LIN {X 0,Y 301.747,Z 438.159,A -85,B 0,C 180,E1 -16541.674,E2 -16541.674} C_VEL
LIN {X 0,Y 303.087,Z 433.963,A -85,B 0,C 180,E1 -16543.844,E2 -16543.844} C_VEL
LIN {X 0,Y 304.497,Z 429.034,A -85,B 0,C 180,E1 -16545.781,E2 -16545.781} C_VEL
LIN {X 0,Y 306.519,Z 421.411,A -85,B 0,C 180,E1 -16548.091,E2 -16548.091} C_VEL
LIN {X 0,Y 308.265,Z 414.22,A -85,B 0,C 180,E1 -16549.823,E2 -16549.823} C_VEL
LIN {X 0,Y 310.172,Z 405.497,A -85,B 0,C 180,E1 -16551.531,E2 -16551.531} C_VEL
LIN {X 0,Y 312.108,Z 395.019,A -85,B 0,C 180,E1 -16553.171,E2 -16553.171} C_VEL
LIN {X 0,Y 312.343,Z 393.686,A -85,B 0,C 180,E1 -16553.358,E2 -16553.358} C_VEL
LIN {X 0,Y 310.159,Z 384.516,A -85,B 0,C 180,E1 -16554.99,E2 -16554.99} C_VEL
LIN {X 0,Y 307.115,Z 376.232,A -85,B 0,C 180,E1 -16556.443,E2 -16556.443} C_VEL
LIN {X 0,Y 305.388,Z 373.91,A -85,B 0,C 180,E1 -16556.951,E2 -16556.951} C_VEL
LIN {X 0,Y 301.445,Z 371.285,A -85,B 0,C 180,E1 -16557.846,E2 -16557.846} C_VEL
LIN {X 0,Y 297.397,Z 368.735,A -85,B 0,C 180,E1 -16558.76,E2 -16558.76} C_VEL
LIN {X 0,Y 295.474,Z 366.51,A -85,B 0,C 180,E1 -16559.287,E2 -16559.287} C_VEL
LIN {X 0,Y 292.034,Z 359.85,A -85,B 0,C 180,E1 -16560.517,E2 -16560.517} C_VEL
LIN {X 0,Y 291.896,Z 359.149,A -85,B 0,C 180,E1 -16560.949,E2 -16560.949} C_VEL
LIN {X 0,Y 291.539,Z 359.172,A -85,B 0,C 180,E1 -16564.147,E2 -16564.147} C_VEL
LIN {X 0,Y 291.714,Z 359.147,A -85,B 0,C 180,E1 -16566.919,E2 -16566.919} C_VEL
LIN {X 0,Y 291.561,Z 359.165,A -85,B 0,C 180,E1 -16569.714,E2 -16569.714} C_VEL
LIN {X 0,Y 291.508,Z 359.173,A -85,B 0,C 180,E1 -16573.951,E2 -16573.951} C_VEL
LIN {X 0,Y 291.426,Z 359.18,A -85,B 0,C 180,E1 -16576.822,E2 -16576.822} C_VEL
LIN {X 0,Y 291.418,Z 359.182,A -85,B 0,C 180,E1 -16579.861,E2 -16579.861} C_VEL
LIN {X 0,Y 291.376,Z 359.185,A -85,B 0,C 180,E1 -16584.208,E2 -16584.208} C_VEL
LIN {X 0,Y 291.413,Z 359.184,A -85,B 0,C 180,E1 -16587.273,E2 -16587.273} C_VEL
LIN {X 0,Y 291.329,Z 359.196,A -85,B 0,C 180,E1 -16590.438,E2 -16590.438} C_VEL
LIN {X 0,Y 291.381,Z 359.44,A -85,B 0,C 180,E1 -16593.337,E2 -16593.337} C_VEL
LIN {X 0,Y 292.227,Z 363.097,A -85,B 0,C 180,E1 -16596.959,E2 -16596.959} C_VEL
LIN {X 0,Y 293.339,Z 368.291,A -85,B 0,C 180,E1 -16601.213,E2 -16601.213} C_VEL
LIN {X 0,Y 294.41,Z 373.527,A -85,B 0,C 180,E1 -16604.848,E2 -16604.848} C_VEL
LIN {X 0,Y 295.479,Z 379.098,A -85,B 0,C 180,E1 -16608.244,E2 -16608.244} C_VEL
LIN {X 0,Y 296.242,Z 383.983,A -85,B 0,C 180,E1 -16610.941,E2 -16610.941} C_VEL
LIN {X 0,Y 296.147,Z 385.908,A -85,B 0,C 180,E1 -16611.902,E2 -16611.902} C_VEL
LIN {X 0,Y 294.347,Z 394.571,A -85,B 0,C 180,E1 -16615.869,E2 -16615.869} C_VEL
LIN {X 0,Y 292.656,Z 405.269,A -85,B 0,C 180,E1 -16620.509,E2 -16620.509} C_VEL
LIN {X 0,Y 292.601,Z 406.741,A -85,B 0,C 180,E1 -16620.947,E2 -16620.947} C_VEL
LIN {X 0,Y 296.051,Z 421.846,A -85,B 0,C 180,E1 -16622.426,E2 -16622.426} C_VEL
LIN {X 0,Y 298.005,Z 434.056,A -85,B 0,C 180,E1 -16623.66,E2 -16623.66} C_VEL
LIN {X 0,Y 298.946,Z 446.03,A -85,B 0,C 180,E1 -16624.966,E2 -16624.966} C_VEL
LIN {X 0,Y 298.863,Z 458.909,A -85,B 0,C 180,E1 -16626.508,E2 -16626.508} C_VEL
LIN {X 0,Y 297.735,Z 470.963,A -85,B 0,C 180,E1 -16628.175,E2 -16628.175} C_VEL
LIN {X 0,Y 296.455,Z 481.364,A -85,B 0,C 180,E1 -16629.895,E2 -16629.895} C_VEL
LIN {X 0,Y 294.247,Z 491.64,A -85,B 0,C 180,E1 -16631.911,E2 -16631.911} C_VEL
LIN {X 0,Y 292.426,Z 500.348,A -85,B 0,C 180,E1 -16634.016,E2 -16634.016} C_VEL
LIN {X 0,Y 291.545,Z 506.044,A -85,B 0,C 180,E1 -16635.695,E2 -16635.695} C_VEL
LIN {X 0,Y 290.556,Z 512.87,A -85,B 0,C 180,E1 -16638.136,E2 -16638.136} C_VEL
LIN {X 0,Y 290.137,Z 517.474,A -85,B 0,C 180,E1 -16640.238,E2 -16640.238} C_VEL
LIN {X 0,Y 290.167,Z 521.068,A -85,B 0,C 180,E1 -16642.345,E2 -16642.345} C_VEL
LIN {X 0,Y 290.425,Z 523.677,A -85,B 0,C 180,E1 -16644.445,E2 -16644.445} C_VEL
LIN {X 0,Y 290.726,Z 524.917,A -85,B 0,C 180,E1 -16645.841,E2 -16645.841} C_VEL
LIN {X 0,Y 291.329,Z 526.05,A -85,B 0,C 180,E1 -16648.618,E2 -16648.618} C_VEL
LIN {X 0,Y 291.637,Z 525.995,A -85,B 0,C 180,E1 -16650,E2 -16650} C_VEL
LIN {X 0,Y 291.369,Z 525.423,A -85,B 0,C 180,E1 -16651.382,E2 -16651.382} C_VEL
LIN {X 0,Y 291.047,Z 524.355,A -85,B 0,C 180,E1 -16652.768,E2 -16652.768} C_VEL
LIN {X 0,Y 290.904,Z 522.87,A -85,B 0,C 180,E1 -16654.156,E2 -16654.156} C_VEL
LIN {X 0,Y 290.642,Z 519.728,A -85,B 0,C 180,E1 -16656.247,E2 -16656.247} C_VEL
LIN {X 0,Y 290.456,Z 515.429,A -85,B 0,C 180,E1 -16658.347,E2 -16658.347} C_VEL
LIN {X 0,Y 290.489,Z 509.882,A -85,B 0,C 180,E1 -16660.454,E2 -16660.454} C_VEL
LIN {X 0,Y 290.897,Z 502.911,A -85,B 0,C 180,E1 -16662.558,E2 -16662.558} C_VEL
LIN {X 0,Y 291.721,Z 494.208,A -85,B 0,C 180,E1 -16664.652,E2 -16664.652} C_VEL
LIN {X 0,Y 292.782,Z 485.266,A -85,B 0,C 180,E1 -16666.399,E2 -16666.399} C_VEL
LIN {X 0,Y 293.913,Z 475.665,A -85,B 0,C 180,E1 -16667.93,E2 -16667.93} C_VEL
LIN {X 0,Y 293.764,Z 463.078,A -85,B 0,C 180,E1 -16669.568,E2 -16669.568} C_VEL
LIN {X 0,Y 293.258,Z 451.021,A -85,B 0,C 180,E1 -16670.828,E2 -16670.828} C_VEL
LIN {X 0,Y 292.555,Z 438.329,A -85,B 0,C 180,E1 -16671.86,E2 -16671.86} C_VEL
LIN {X 0,Y 291.466,Z 424.734,A -85,B 0,C 180,E1 -16672.693,E2 -16672.693} C_VEL
LIN {X 0,Y 290.934,Z 418.518,A -85,B 0,C 180,E1 -16673.031,E2 -16673.031} C_VEL
LIN {X 0,Y 291.153,Z 415.339,A -85,B 0,C 180,E1 -16674.226,E2 -16674.226} C_VEL
LIN {X 0,Y 292.285,Z 404.281,A -85,B 0,C 180,E1 -16678.743,E2 -16678.743} C_VEL
LIN {X 0,Y 293.696,Z 393.683,A -85,B 0,C 180,E1 -16683.119,E2 -16683.119} C_VEL
LIN {X 0,Y 295.372,Z 383.621,A -85,B 0,C 180,E1 -16687.353,E2 -16687.353} C_VEL
LIN {X 0,Y 295.557,Z 381.391,A -85,B 0,C 180,E1 -16688.307,E2 -16688.307} C_VEL
LIN {X 0,Y 294.425,Z 374.995,A -85,B 0,C 180,E1 -16691.223,E2 -16691.223} C_VEL
LIN {X 0,Y 292.932,Z 367.204,A -85,B 0,C 180,E1 -16694.947,E2 -16694.947} C_VEL
LIN {X 0,Y 291.334,Z 359.27,A -85,B 0,C 180,E1 -16698.995,E2 -16698.995} C_VEL
LIN {X 0,Y 291.396,Z 359.188,A -85,B 0,C 180,E1 -16702.918,E2 -16702.918} C_VEL
LIN {X 0,Y 291.34,Z 359.192,A -85,B 0,C 180,E1 -16706.301,E2 -16706.301} C_VEL
LIN {X 0,Y 291.382,Z 359.186,A -85,B 0,C 180,E1 -16710.26,E2 -16710.26} C_VEL
LIN {X 0,Y 291.405,Z 359.184,A -85,B 0,C 180,E1 -16714.271,E2 -16714.271} C_VEL
LIN {X 0,Y 291.366,Z 359.191,A -85,B 0,C 180,E1 -16717.298,E2 -16717.298} C_VEL
LIN {X 0,Y 291.433,Z 359.18,A -85,B 0,C 180,E1 -16720.268,E2 -16720.268} C_VEL
LIN {X 0,Y 291.491,Z 359.175,A -85,B 0,C 180,E1 -16724.665,E2 -16724.665} C_VEL
LIN {X 0,Y 291.521,Z 359.172,A -85,B 0,C 180,E1 -16728.88,E2 -16728.88} C_VEL
LIN {X 0,Y 291.659,Z 359.152,A -85,B 0,C 180,E1 -16731.687,E2 -16731.687} C_VEL
LIN {X 0,Y 291.61,Z 359.16,A -85,B 0,C 180,E1 -16734.468,E2 -16734.468} C_VEL
LIN {X 0,Y 291.881,Z 359.127,A -85,B 0,C 180,E1 -16738.62,E2 -16738.62} C_VEL
LIN {X 0,Y 291.881,Z 359.125,A -85,B 0,C 180,E1 -16741.38,E2 -16741.38} C_VEL
LIN {X 0,Y 291.734,Z 359.146,A -85,B 0,C 180,E1 -16746.918,E2 -16746.918} C_VEL
LIN {X 0,Y 291.622,Z 359.156,A -85,B 0,C 180,E1 -16749.712,E2 -16749.712} C_VEL
LIN {X 0,Y 291.515,Z 359.169,A -85,B 0,C 180,E1 -16753.951,E2 -16753.951} C_VEL
LIN {X 0,Y 291.48,Z 359.177,A -85,B 0,C 180,E1 -16756.818,E2 -16756.818} C_VEL
LIN {X 0,Y 291.445,Z 359.179,A -85,B 0,C 180,E1 -16759.875,E2 -16759.875} C_VEL
LIN {X 0,Y 291.394,Z 359.187,A -85,B 0,C 180,E1 -16764.206,E2 -16764.206} C_VEL
LIN {X 0,Y 291.417,Z 359.182,A -85,B 0,C 180,E1 -16767.272,E2 -16767.272} C_VEL
LIN {X 0,Y 291.332,Z 359.197,A -85,B 0,C 180,E1 -16770.437,E2 -16770.437} C_VEL
LIN {X 0,Y 291.34,Z 359.192,A -85,B 0,C 180,E1 -16773.699,E2 -16773.699} C_VEL
LIN {X 0,Y 291.393,Z 359.184,A -85,B 0,C 180,E1 -16777.26,E2 -16777.26} C_VEL
LIN {X 0,Y 291.372,Z 359.19,A -85,B 0,C 180,E1 -16780.636,E2 -16780.636} C_VEL
LIN {X 0,Y 291.297,Z 359.2,A -85,B 0,C 180,E1 -16784.401,E2 -16784.401} C_VEL
LIN {X 0,Y 291.324,Z 359.196,A -85,B 0,C 180,E1 -16788.405,E2 -16788.405} C_VEL
LIN {X 0,Y 291.362,Z 359.189,A -85,B 0,C 180,E1 -16791.161,E2 -16791.161} C_VEL
LIN {X 0,Y 291.361,Z 359.189,A -85,B 0,C 180,E1 -16794.627,E2 -16794.627} C_VEL
LIN {X 0,Y 291.375,Z 359.192,A -85,B 0,C 180,E1 -16797.952,E2 -16797.952} C_VEL
LIN {X 0,Y 291.387,Z 359.186,A -85,B 0,C 180,E1 -16801.16,E2 -16801.16} C_VEL
LIN {X 0,Y 291.418,Z 359.184,A -85,B 0,C 180,E1 -16804.273,E2 -16804.273} C_VEL
LIN {X 0,Y 291.382,Z 359.187,A -85,B 0,C 180,E1 -16807.3,E2 -16807.3} C_VEL
LIN {X 0,Y 291.459,Z 359.178,A -85,B 0,C 180,E1 -16810.271,E2 -16810.271} C_VEL
LIN {X 0,Y 291.556,Z 359.165,A -85,B 0,C 180,E1 -16814.624,E2 -16814.624} C_VEL
LIN {X 0,Y 291.539,Z 359.166,A -85,B 0,C 180,E1 -16818.881,E2 -16818.881} C_VEL
LIN {X 0,Y 291.712,Z 359.15,A -85,B 0,C 180,E1 -16821.689,E2 -16821.689} C_VEL
LIN {X 0,Y 291.634,Z 359.155,A -85,B 0,C 180,E1 -16824.469,E2 -16824.469} C_VEL
LIN {X 0,Y 291.895,Z 359.122,A -85,B 0,C 180,E1 -16828.62,E2 -16828.62} C_VEL
LIN {X 0,Y 291.892,Z 359.127,A -85,B 0,C 180,E1 -16831.38,E2 -16831.38} C_VEL
LIN {X 0,Y 291.738,Z 359.143,A -85,B 0,C 180,E1 -16836.918,E2 -16836.918} C_VEL
LIN {X 0,Y 291.63,Z 359.158,A -85,B 0,C 180,E1 -16839.712,E2 -16839.712} C_VEL
LIN {X 0,Y 291.524,Z 359.17,A -85,B 0,C 180,E1 -16843.95,E2 -16843.95} C_VEL
LIN {X 0,Y 291.488,Z 359.174,A -85,B 0,C 180,E1 -16846.817,E2 -16846.817} C_VEL
LIN {X 0,Y 291.451,Z 359.179,A -85,B 0,C 180,E1 -16849.874,E2 -16849.874} C_VEL
LIN {X 0,Y 291.399,Z 359.184,A -85,B 0,C 180,E1 -16854.205,E2 -16854.205} C_VEL
LIN {X 0,Y 291.418,Z 359.186,A -85,B 0,C 180,E1 -16857.271,E2 -16857.271} C_VEL
LIN {X 0,Y 291.333,Z 359.193,A -85,B 0,C 180,E1 -16860.436,E2 -16860.436} C_VEL
LIN {X 0,Y 291.343,Z 359.193,A -85,B 0,C 180,E1 -16863.698,E2 -16863.698} C_VEL
LIN {X 0,Y 291.404,Z 359.188,A -85,B 0,C 180,E1 -16867.261,E2 -16867.261} C_VEL
LIN {X 0,Y 291.463,Z 359.34,A -85,B 0,C 180,E1 -16870.445,E2 -16870.445} C_VEL
LIN {X 0,Y 291.684,Z 360.374,A -85,B 0,C 180,E1 -16870.68,E2 -16870.68} C_VEL
LIN {X 0,Y 295.511,Z 373.533,A -85,B 0,C 180,E1 -16872.122,E2 -16872.122} C_VEL
LIN {X 0,Y 297.723,Z 381.938,A -85,B 0,C 180,E1 -16873.2,E2 -16873.2} C_VEL
LIN {X 0,Y 297.506,Z 387.452,A -85,B 0,C 180,E1 -16873.904,E2 -16873.904} C_VEL
LIN {X 0,Y 296.304,Z 399.361,A -85,B 0,C 180,E1 -16875.658,E2 -16875.658} C_VEL
LIN {X 0,Y 295.192,Z 408.983,A -85,B 0,C 180,E1 -16877.423,E2 -16877.423} C_VEL
LIN {X 0,Y 294.133,Z 417.653,A -85,B 0,C 180,E1 -16879.375,E2 -16879.375} C_VEL
LIN {X 0,Y 293.327,Z 425.193,A -85,B 0,C 180,E1 -16881.468,E2 -16881.468} C_VEL
LIN {X 0,Y 292.501,Z 432.164,A -85,B 0,C 180,E1 -16883.937,E2 -16883.937} C_VEL
LIN {X 0,Y 292.005,Z 437.44,A -85,B 0,C 180,E1 -16886.388,E2 -16886.388} C_VEL
LIN {X 0,Y 291.744,Z 441.153,A -85,B 0,C 180,E1 -16888.807,E2 -16888.807} C_VEL
LIN {X 0,Y 291.721,Z 443.554,A -85,B 0,C 180,E1 -16891.195,E2 -16891.195} C_VEL
LIN {X 0,Y 291.842,Z 444.59,A -85,B 0,C 180,E1 -16892.998,E2 -16892.998} C_VEL
LIN {X 0,Y 292.048,Z 444.896,A -85,B 0,C 180,E1 -16894.332,E2 -16894.332} C_VEL
LIN {X 0,Y 292.447,Z 444.8,A -85,B 0,C 180,E1 -16895.949,E2 -16895.949} C_VEL
LIN {X 0,Y 292.9,Z 444.204,A -85,B 0,C 180,E1 -16897.424,E2 -16897.424} C_VEL
LIN {X 0,Y 293.512,Z 443.042,A -85,B 0,C 180,E1 -16899.037,E2 -16899.037} C_VEL
LIN {X 0,Y 294.518,Z 440.572,A -85,B 0,C 180,E1 -16901.207,E2 -16901.207} C_VEL
LIN {X 0,Y 295.861,Z 436.851,A -85,B 0,C 180,E1 -16903.438,E2 -16903.438} C_VEL
LIN {X 0,Y 297.42,Z 431.843,A -85,B 0,C 180,E1 -16905.65,E2 -16905.65} C_VEL
LIN {X 0,Y 299.307,Z 425.489,A -85,B 0,C 180,E1 -16907.8,E2 -16907.8} C_VEL
LIN {X 0,Y 301.082,Z 418.897,A -85,B 0,C 180,E1 -16909.58,E2 -16909.58} C_VEL
LIN {X 0,Y 303.008,Z 410.961,A -85,B 0,C 180,E1 -16911.329,E2 -16911.329} C_VEL
LIN {X 0,Y 305.084,Z 401.311,A -85,B 0,C 180,E1 -16913.036,E2 -16913.036} C_VEL
LIN {X 0,Y 305.93,Z 396.746,A -85,B 0,C 180,E1 -16913.736,E2 -16913.736} C_VEL
LIN {X 0,Y 305.723,Z 393.97,A -85,B 0,C 180,E1 -16914.234,E2 -16914.234} C_VEL
LIN {X 0,Y 303.779,Z 386.226,A -85,B 0,C 180,E1 -16915.688,E2 -16915.688} C_VEL
LIN {X 0,Y 300.007,Z 376.53,A -85,B 0,C 180,E1 -16917.499,E2 -16917.499} C_VEL
LIN {X 0,Y 295.799,Z 367.062,A -85,B 0,C 180,E1 -16919.181,E2 -16919.181} C_VEL
LIN {X 0,Y 295.474,Z 366.51,A -85,B 0,C 180,E1 -16919.287,E2 -16919.287} C_VEL
LIN {X 0,Y 293.577,Z 364.13,A -85,B 0,C 180,E1 -16919.839,E2 -16919.839} C_VEL
LIN {X 0,Y 289.506,Z 361.509,A -85,B 0,C 180,E1 -16920.824,E2 -16920.824} C_VEL
LIN {X 0,Y 286.336,Z 360.394,A -85,B 0,C 180,E1 -16921.682,E2 -16921.682} C_VEL
LIN {X 0,Y 284.881,Z 360.039,A -85,B 0,C 180,E1 -16922.422,E2 -16922.422} C_VEL
LIN {X 0,Y 284.743,Z 360.017,A -85,B 0,C 180,E1 -16922.687,E2 -16922.687} C_VEL
LIN {X 0,Y 284.665,Z 360.026,A -85,B 0,C 180,E1 -16927.091,E2 -16927.091} C_VEL
LIN {X 0,Y 284.507,Z 360.044,A -85,B 0,C 180,E1 -16929.958,E2 -16929.958} C_VEL
LIN {X 0,Y 284.456,Z 360.053,A -85,B 0,C 180,E1 -16934.304,E2 -16934.304} C_VEL
LIN {X 0,Y 284.356,Z 360.062,A -85,B 0,C 180,E1 -16938.742,E2 -16938.742} C_VEL
LIN {X 0,Y 284.309,Z 360.068,A -85,B 0,C 180,E1 -16941.765,E2 -16941.765} C_VEL
LIN {X 0,Y 284.33,Z 360.068,A -85,B 0,C 180,E1 -16944.847,E2 -16944.847} C_VEL
LIN {X 0,Y 284.322,Z 360.068,A -85,B 0,C 180,E1 -16948.012,E2 -16948.012} C_VEL
LIN {X 0,Y 284.322,Z 360.288,A -85,B 0,C 180,E1 -16951.683,E2 -16951.683} C_VEL
LIN {X 0,Y 285.149,Z 363.846,A -85,B 0,C 180,E1 -16955.578,E2 -16955.578} C_VEL
LIN {X 0,Y 286.14,Z 368.455,A -85,B 0,C 180,E1 -16959.687,E2 -16959.687} C_VEL
LIN {X 0,Y 287.406,Z 374.342,A -85,B 0,C 180,E1 -16964.057,E2 -16964.057} C_VEL
LIN {X 0,Y 288.542,Z 380.473,A -85,B 0,C 180,E1 -16967.962,E2 -16967.962} C_VEL
LIN {X 0,Y 289.336,Z 385.842,A -85,B 0,C 180,E1 -16971.013,E2 -16971.013} C_VEL
LIN {X 0,Y 288.834,Z 388.945,A -85,B 0,C 180,E1 -16972.534,E2 -16972.534} C_VEL
LIN {X 0,Y 286.927,Z 398.192,A -85,B 0,C 180,E1 -16976.845,E2 -16976.845} C_VEL
LIN {X 0,Y 285.916,Z 404.822,A -85,B 0,C 180,E1 -16979.691,E2 -16979.691} C_VEL
LIN {X 0,Y 286.502,Z 408.028,A -85,B 0,C 180,E1 -16980.074,E2 -16980.074} C_VEL
LIN {X 0,Y 289.27,Z 418.993,A -85,B 0,C 180,E1 -16981.228,E2 -16981.228} C_VEL
LIN {X 0,Y 291.495,Z 433.005,A -85,B 0,C 180,E1 -16982.737,E2 -16982.737} C_VEL
LIN {X 0,Y 292.615,Z 446.26,A -85,B 0,C 180,E1 -16984.261,E2 -16984.261} C_VEL
LIN {X 0,Y 292.378,Z 458.983,A -85,B 0,C 180,E1 -16985.882,E2 -16985.882} C_VEL
LIN {X 0,Y 291.136,Z 471.212,A -85,B 0,C 180,E1 -16987.654,E2 -16987.654} C_VEL
LIN {X 0,Y 289.735,Z 481.334,A -85,B 0,C 180,E1 -16989.408,E2 -16989.408} C_VEL
LIN {X 0,Y 287.824,Z 489.848,A -85,B 0,C 180,E1 -16991.124,E2 -16991.124} C_VEL
LIN {X 0,Y 285.862,Z 498.805,A -85,B 0,C 180,E1 -16993.328,E2 -16993.328} C_VEL
LIN {X 0,Y 284.389,Z 506.549,A -85,B 0,C 180,E1 -16995.693,E2 -16995.693} C_VEL
LIN {X 0,Y 283.539,Z 512.172,A -85,B 0,C 180,E1 -16997.838,E2 -16997.838} C_VEL
LIN {X 0,Y 283.086,Z 516.691,A -85,B 0,C 180,E1 -16999.992,E2 -16999.992} C_VEL
LIN {X 0,Y 283.185,Z 521.141,A -85,B 0,C 180,E1 -17002.872,E2 -17002.872} C_VEL
LIN {X 0,Y 283.336,Z 522.751,A -85,B 0,C 180,E1 -17004.306,E2 -17004.306} C_VEL
LIN {X 0,Y 283.637,Z 523.923,A -85,B 0,C 180,E1 -17005.737,E2 -17005.737} C_VEL
LIN {X 0,Y 284.291,Z 524.993,A -85,B 0,C 180,E1 -17008.583,E2 -17008.583} C_VEL
LIN {X 0,Y 284.613,Z 524.907,A -85,B 0,C 180,E1 -17010,E2 -17010} C_VEL
LIN {X 0,Y 284.337,Z 524.26,A -85,B 0,C 180,E1 -17011.416,E2 -17011.416} C_VEL
LIN {X 0,Y 284.013,Z 523.149,A -85,B 0,C 180,E1 -17012.837,E2 -17012.837} C_VEL
LIN {X 0,Y 283.786,Z 520.672,A -85,B 0,C 180,E1 -17014.972,E2 -17014.972} C_VEL
LIN {X 0,Y 283.486,Z 516.504,A -85,B 0,C 180,E1 -17017.406,E2 -17017.406} C_VEL
LIN {X 0,Y 283.37,Z 512.259,A -85,B 0,C 180,E1 -17019.277,E2 -17019.277} C_VEL
LIN {X 0,Y 283.621,Z 506.169,A -85,B 0,C 180,E1 -17021.434,E2 -17021.434} C_VEL
LIN {X 0,Y 284.242,Z 498.554,A -85,B 0,C 180,E1 -17023.585,E2 -17023.585} C_VEL
LIN {X 0,Y 285.017,Z 490.762,A -85,B 0,C 180,E1 -17025.371,E2 -17025.371} C_VEL
LIN {X 0,Y 286.295,Z 480.316,A -85,B 0,C 180,E1 -17027.316,E2 -17027.316} C_VEL
LIN {X 0,Y 286.801,Z 474.664,A -85,B 0,C 180,E1 -17028.206,E2 -17028.206} C_VEL
LIN {X 0,Y 286.728,Z 463.614,A -85,B 0,C 180,E1 -17029.695,E2 -17029.695} C_VEL
LIN {X 0,Y 286.233,Z 450.892,A -85,B 0,C 180,E1 -17031.087,E2 -17031.087} C_VEL
LIN {X 0,Y 285.57,Z 438.57,A -85,B 0,C 180,E1 -17032.138,E2 -17032.138} C_VEL
LIN {X 0,Y 284.449,Z 424.061,A -85,B 0,C 180,E1 -17033.069,E2 -17033.069} C_VEL
LIN {X 0,Y 283.947,Z 417.569,A -85,B 0,C 180,E1 -17033.439,E2 -17033.439} C_VEL
LIN {X 0,Y 284.578,Z 410.324,A -85,B 0,C 180,E1 -17036.393,E2 -17036.393} C_VEL
LIN {X 0,Y 285.889,Z 399.224,A -85,B 0,C 180,E1 -17041.08,E2 -17041.08} C_VEL
LIN {X 0,Y 287.327,Z 389.837,A -85,B 0,C 180,E1 -17045.085,E2 -17045.085} C_VEL
LIN {X 0,Y 288.491,Z 382.8,A -85,B 0,C 180,E1 -17048.135,E2 -17048.135} C_VEL
LIN {X 0,Y 287.939,Z 378.685,A -85,B 0,C 180,E1 -17050.047,E2 -17050.047} C_VEL
LIN {X 0,Y 286.118,Z 369.319,A -85,B 0,C 180,E1 -17054.575,E2 -17054.575} C_VEL
LIN {X 0,Y 284.701,Z 362.214,A -85,B 0,C 180,E1 -17058.202,E2 -17058.202} C_VEL
LIN {X 0,Y 284.29,Z 360.123,A -85,B 0,C 180,E1 -17059.422,E2 -17059.422} C_VEL
LIN {X 0,Y 284.322,Z 360.069,A -85,B 0,C 180,E1 -17063.612,E2 -17063.612} C_VEL
LIN {X 0,Y 284.303,Z 360.073,A -85,B 0,C 180,E1 -17067.189,E2 -17067.189} C_VEL
LIN {X 0,Y 284.354,Z 360.062,A -85,B 0,C 180,E1 -17070.375,E2 -17070.375} C_VEL
LIN {X 0,Y 284.369,Z 360.062,A -85,B 0,C 180,E1 -17073.586,E2 -17073.586} C_VEL
LIN {X 0,Y 284.327,Z 360.066,A -85,B 0,C 180,E1 -17076.703,E2 -17076.703} C_VEL
LIN {X 0,Y 284.37,Z 360.06,A -85,B 0,C 180,E1 -17079.904,E2 -17079.904} C_VEL
LIN {X 0,Y 284.44,Z 360.052,A -85,B 0,C 180,E1 -17084.492,E2 -17084.492} C_VEL
LIN {X 0,Y 284.459,Z 360.049,A -85,B 0,C 180,E1 -17088.6,E2 -17088.6} C_VEL
LIN {X 0,Y 284.614,Z 360.031,A -85,B 0,C 180,E1 -17091.48,E2 -17091.48} C_VEL
LIN {X 0,Y 284.58,Z 360.035,A -85,B 0,C 180,E1 -17094.331,E2 -17094.331} C_VEL
LIN {X 0,Y 284.847,Z 360.003,A -85,B 0,C 180,E1 -17098.586,E2 -17098.586} C_VEL
LIN {X 0,Y 284.847,Z 360.001,A -85,B 0,C 180,E1 -17101.414,E2 -17101.414} C_VEL
LIN {X 0,Y 284.686,Z 360.022,A -85,B 0,C 180,E1 -17107.09,E2 -17107.09} C_VEL
LIN {X 0,Y 284.56,Z 360.037,A -85,B 0,C 180,E1 -17109.956,E2 -17109.956} C_VEL
LIN {X 0,Y 284.471,Z 360.049,A -85,B 0,C 180,E1 -17114.303,E2 -17114.303} C_VEL
LIN {X 0,Y 284.419,Z 360.054,A -85,B 0,C 180,E1 -17117.249,E2 -17117.249} C_VEL
LIN {X 0,Y 284.373,Z 360.062,A -85,B 0,C 180,E1 -17120.243,E2 -17120.243} C_VEL
LIN {X 0,Y 284.363,Z 360.061,A -85,B 0,C 180,E1 -17123.876,E2 -17123.876} C_VEL
LIN {X 0,Y 284.392,Z 360.057,A -85,B 0,C 180,E1 -17127.174,E2 -17127.174} C_VEL
LIN {X 0,Y 284.29,Z 360.069,A -85,B 0,C 180,E1 -17131.275,E2 -17131.275} C_VEL
LIN {X 0,Y 284.357,Z 360.061,A -85,B 0,C 180,E1 -17135.355,E2 -17135.355} C_VEL
LIN {X 0,Y 284.325,Z 360.069,A -85,B 0,C 180,E1 -17138.167,E2 -17138.167} C_VEL
LIN {X 0,Y 284.298,Z 360.071,A -85,B 0,C 180,E1 -17141.871,E2 -17141.871} C_VEL
LIN {X 0,Y 284.254,Z 360.078,A -85,B 0,C 180,E1 -17146.19,E2 -17146.19} C_VEL
LIN {X 0,Y 284.305,Z 360.072,A -85,B 0,C 180,E1 -17150.025,E2 -17150.025} C_VEL
LIN {X 0,Y 284.335,Z 360.066,A -85,B 0,C 180,E1 -17153.616,E2 -17153.616} C_VEL
LIN {X 0,Y 284.308,Z 360.068,A -85,B 0,C 180,E1 -17157.19,E2 -17157.19} C_VEL
LIN {X 0,Y 284.362,Z 360.062,A -85,B 0,C 180,E1 -17160.377,E2 -17160.377} C_VEL
LIN {X 0,Y 284.379,Z 360.06,A -85,B 0,C 180,E1 -17163.587,E2 -17163.587} C_VEL
LIN {X 0,Y 284.367,Z 360.06,A -85,B 0,C 180,E1 -17166.708,E2 -17166.708} C_VEL
LIN {X 0,Y 284.405,Z 360.056,A -85,B 0,C 180,E1 -17171.262,E2 -17171.262} C_VEL
LIN {X 0,Y 284.493,Z 360.045,A -85,B 0,C 180,E1 -17174.459,E2 -17174.459} C_VEL
LIN {X 0,Y 284.49,Z 360.044,A -85,B 0,C 180,E1 -17178.602,E2 -17178.602} C_VEL
LIN {X 0,Y 284.662,Z 360.026,A -85,B 0,C 180,E1 -17181.481,E2 -17181.481} C_VEL
LIN {X 0,Y 284.604,Z 360.031,A -85,B 0,C 180,E1 -17184.331,E2 -17184.331} C_VEL
LIN {X 0,Y 284.861,Z 359.999,A -85,B 0,C 180,E1 -17188.586,E2 -17188.586} C_VEL
LIN {X 0,Y 284.858,Z 360.003,A -85,B 0,C 180,E1 -17191.414,E2 -17191.414} C_VEL
LIN {X 0,Y 284.69,Z 360.021,A -85,B 0,C 180,E1 -17197.09,E2 -17197.09} C_VEL
LIN {X 0,Y 284.568,Z 360.036,A -85,B 0,C 180,E1 -17199.955,E2 -17199.955} C_VEL
LIN {X 0,Y 284.483,Z 360.046,A -85,B 0,C 180,E1 -17204.302,E2 -17204.302} C_VEL
LIN {X 0,Y 284.426,Z 360.057,A -85,B 0,C 180,E1 -17207.248,E2 -17207.248} C_VEL
LIN {X 0,Y 284.379,Z 360.059,A -85,B 0,C 180,E1 -17210.242,E2 -17210.242} C_VEL
LIN {X 0,Y 284.369,Z 360.061,A -85,B 0,C 180,E1 -17213.875,E2 -17213.875} C_VEL
LIN {X 0,Y 284.394,Z 360.062,A -85,B 0,C 180,E1 -17217.172,E2 -17217.172} C_VEL
LIN {X 0,Y 284.293,Z 360.074,A -85,B 0,C 180,E1 -17221.274,E2 -17221.274} C_VEL
LIN {X 0,Y 284.361,Z 360.065,A -85,B 0,C 180,E1 -17225.353,E2 -17225.353} C_VEL
LIN {X 0,Y 284.337,Z 360.066,A -85,B 0,C 180,E1 -17228.164,E2 -17228.164} C_VEL
LIN {X 0,Y 284.408,Z 360.225,A -85,B 0,C 180,E1 -17230.06,E2 -17230.06} C_VEL
LIN {X 0,Y 284.644,Z 361.282,A -85,B 0,C 180,E1 -17230.311,E2 -17230.311} C_VEL
LIN {X 0,Y 288.442,Z 374.248,A -85,B 0,C 180,E1 -17231.761,E2 -17231.761} C_VEL
LIN {X 0,Y 290.894,Z 383.724,A -85,B 0,C 180,E1 -17233.019,E2 -17233.019} C_VEL
LIN {X 0,Y 289.968,Z 394.558,A -85,B 0,C 180,E1 -17234.503,E2 -17234.503} C_VEL
LIN {X 0,Y 288.875,Z 404.197,A -85,B 0,C 180,E1 -17236.102,E2 -17236.102} C_VEL
LIN {X 0,Y 287.849,Z 412.764,A -85,B 0,C 180,E1 -17237.822,E2 -17237.822} C_VEL
LIN {X 0,Y 286.84,Z 421.108,A -85,B 0,C 180,E1 -17239.881,E2 -17239.881} C_VEL
LIN {X 0,Y 286,Z 428.357,A -85,B 0,C 180,E1 -17242.096,E2 -17242.096} C_VEL
LIN {X 0,Y 285.347,Z 434.275,A -85,B 0,C 180,E1 -17244.366,E2 -17244.366} C_VEL
LIN {X 0,Y 284.979,Z 438.227,A -85,B 0,C 180,E1 -17246.298,E2 -17246.298} C_VEL
LIN {X 0,Y 284.725,Z 442.042,A -85,B 0,C 180,E1 -17248.778,E2 -17248.778} C_VEL
LIN {X 0,Y 284.656,Z 443.831,A -85,B 0,C 180,E1 -17250.41,E2 -17250.41} C_VEL
LIN {X 0,Y 284.796,Z 445.425,A -85,B 0,C 180,E1 -17252.668,E2 -17252.668} C_VEL
LIN {X 0,Y 285.357,Z 445.961,A -85,B 0,C 180,E1 -17255.677,E2 -17255.677} C_VEL
LIN {X 0,Y 286.264,Z 444.911,A -85,B 0,C 180,E1 -17258.392,E2 -17258.392} C_VEL
LIN {X 0,Y 286.911,Z 443.626,A -85,B 0,C 180,E1 -17259.944,E2 -17259.944} C_VEL
LIN {X 0,Y 288.024,Z 440.999,A -85,B 0,C 180,E1 -17262.102,E2 -17262.102} C_VEL
LIN {X 0,Y 289.61,Z 436.747,A -85,B 0,C 180,E1 -17264.518,E2 -17264.518} C_VEL
LIN {X 0,Y 291.436,Z 431.42,A -85,B 0,C 180,E1 -17266.756,E2 -17266.756} C_VEL
LIN {X 0,Y 293.526,Z 424.414,A -85,B 0,C 180,E1 -17269.008,E2 -17269.008} C_VEL
LIN {X 0,Y 295.826,Z 416.09,A -85,B 0,C 180,E1 -17271.117,E2 -17271.117} C_VEL
LIN {X 0,Y 298.037,Z 406.969,A -85,B 0,C 180,E1 -17272.946,E2 -17272.946} C_VEL
LIN {X 0,Y 299.782,Z 398.342,A -85,B 0,C 180,E1 -17274.369,E2 -17274.369} C_VEL
LIN {X 0,Y 298.129,Z 390.346,A -85,B 0,C 180,E1 -17275.945,E2 -17275.945} C_VEL
LIN {X 0,Y 295.454,Z 382.751,A -85,B 0,C 180,E1 -17277.482,E2 -17277.482} C_VEL
LIN {X 0,Y 291.417,Z 372.819,A -85,B 0,C 180,E1 -17279.374,E2 -17279.374} C_VEL
LIN {X 0,Y 287.018,Z 364.261,A -85,B 0,C 180,E1 -17281.052,E2 -17281.052} C_VEL
LIN {X 0,Y 285.858,Z 362.838,A -85,B 0,C 180,E1 -17281.409,E2 -17281.409} C_VEL
LIN {X 0,Y 284.899,Z 360.633,A -85,B 0,C 180,E1 -17281.855,E2 -17281.855} C_VEL
LIN {X 0,Y 284.766,Z 360.035,A -85,B 0,C 180,E1 -17282.299,E2 -17282.299} C_VEL
LIN {X 0,Y 284.743,Z 360.017,A -85,B 0,C 180,E1 -17282.687,E2 -17282.687} C_VEL
LIN {X 0,Y 284.014,Z 360.116,A -85,B 0,C 180,E1 -17283.866,E2 -17283.866} C_VEL
LIN {X 0,Y 281.121,Z 360.472,A -85,B 0,C 180,E1 -17285.786,E2 -17285.786} C_VEL
LIN {X 0,Y 278.695,Z 360.772,A -85,B 0,C 180,E1 -17287.345,E2 -17287.345} C_VEL
LIN {X 0,Y 277.648,Z 360.899,A -85,B 0,C 180,E1 -17288.554,E2 -17288.554} C_VEL
LIN {X 0,Y 277.557,Z 360.912,A -85,B 0,C 180,E1 -17288.963,E2 -17288.963} C_VEL
LIN {X 0,Y 277.402,Z 360.931,A -85,B 0,C 180,E1 -17293.18,E2 -17293.18} C_VEL
LIN {X 0,Y 277.353,Z 360.938,A -85,B 0,C 180,E1 -17296.185,E2 -17296.185} C_VEL
LIN {X 0,Y 277.307,Z 360.935,A -85,B 0,C 180,E1 -17300.332,E2 -17300.332} C_VEL
LIN {X 0,Y 277.286,Z 360.939,A -85,B 0,C 180,E1 -17304.158,E2 -17304.158} C_VEL
LIN {X 0,Y 277.318,Z 360.942,A -85,B 0,C 180,E1 -17307.504,E2 -17307.504} C_VEL
LIN {X 0,Y 277.332,Z 360.993,A -85,B 0,C 180,E1 -17309.614,E2 -17309.614} C_VEL
LIN {X 0,Y 277.987,Z 364.382,A -85,B 0,C 180,E1 -17313.793,E2 -17313.793} C_VEL
LIN {X 0,Y 278.743,Z 367.81,A -85,B 0,C 180,E1 -17317.237,E2 -17317.237} C_VEL
LIN {X 0,Y 279.731,Z 372.332,A -85,B 0,C 180,E1 -17321.088,E2 -17321.088} C_VEL
LIN {X 0,Y 280.711,Z 377.002,A -85,B 0,C 180,E1 -17324.509,E2 -17324.509} C_VEL
LIN {X 0,Y 281.835,Z 383.092,A -85,B 0,C 180,E1 -17328.426,E2 -17328.426} C_VEL
LIN {X 0,Y 282.376,Z 386.655,A -85,B 0,C 180,E1 -17330.494,E2 -17330.494} C_VEL
LIN {X 0,Y 282.308,Z 388.542,A -85,B 0,C 180,E1 -17331.512,E2 -17331.512} C_VEL
LIN {X 0,Y 280.313,Z 397.455,A -85,B 0,C 180,E1 -17335.831,E2 -17335.831} C_VEL
LIN {X 0,Y 279.321,Z 403.25,A -85,B 0,C 180,E1 -17338.409,E2 -17338.409} C_VEL
LIN {X 0,Y 279.955,Z 406.639,A -85,B 0,C 180,E1 -17338.832,E2 -17338.832} C_VEL
LIN {X 0,Y 281.908,Z 413.565,A -85,B 0,C 180,E1 -17339.643,E2 -17339.643} C_VEL
LIN {X 0,Y 284.617,Z 427.67,A -85,B 0,C 180,E1 -17341.243,E2 -17341.243} C_VEL
LIN {X 0,Y 285.977,Z 440.552,A -85,B 0,C 180,E1 -17342.778,E2 -17342.778} C_VEL
LIN {X 0,Y 286.252,Z 452.88,A -85,B 0,C 180,E1 -17344.36,E2 -17344.36} C_VEL
LIN {X 0,Y 285.554,Z 463.595,A -85,B 0,C 180,E1 -17345.867,E2 -17345.867} C_VEL
LIN {X 0,Y 284.054,Z 474.626,A -85,B 0,C 180,E1 -17347.642,E2 -17347.642} C_VEL
LIN {X 0,Y 282.321,Z 484.79,A -85,B 0,C 180,E1 -17349.604,E2 -17349.604} C_VEL
LIN {X 0,Y 280.041,Z 494.025,A -85,B 0,C 180,E1 -17351.718,E2 -17351.718} C_VEL
LIN {X 0,Y 278.236,Z 501.658,A -85,B 0,C 180,E1 -17353.868,E2 -17353.868} C_VEL
LIN {X 0,Y 277.098,Z 507.947,A -85,B 0,C 180,E1 -17356.058,E2 -17356.058} C_VEL
LIN {X 0,Y 276.293,Z 513.078,A -85,B 0,C 180,E1 -17358.259,E2 -17358.259} C_VEL
LIN {X 0,Y 275.957,Z 517.163,A -85,B 0,C 180,E1 -17360.472,E2 -17360.472} C_VEL
LIN {X 0,Y 276.136,Z 520.662,A -85,B 0,C 180,E1 -17363.026,E2 -17363.026} C_VEL
LIN {X 0,Y 276.552,Z 522.927,A -85,B 0,C 180,E1 -17365.628,E2 -17365.628} C_VEL
LIN {X 0,Y 277.251,Z 523.939,A -85,B 0,C 180,E1 -17368.548,E2 -17368.548} C_VEL
LIN {X 0,Y 277.587,Z 523.801,A -85,B 0,C 180,E1 -17370,E2 -17370} C_VEL
LIN {X 0,Y 277.305,Z 523.094,A -85,B 0,C 180,E1 -17371.452,E2 -17371.452} C_VEL
LIN {X 0,Y 276.976,Z 521.947,A -85,B 0,C 180,E1 -17372.909,E2 -17372.909} C_VEL
LIN {X 0,Y 276.755,Z 519.388,A -85,B 0,C 180,E1 -17375.099,E2 -17375.099} C_VEL
LIN {X 0,Y 276.438,Z 515.369,A -85,B 0,C 180,E1 -17377.468,E2 -17377.468} C_VEL
LIN {X 0,Y 276.336,Z 510.784,A -85,B 0,C 180,E1 -17379.515,E2 -17379.515} C_VEL
LIN {X 0,Y 276.635,Z 504.59,A -85,B 0,C 180,E1 -17381.726,E2 -17381.726} C_VEL
LIN {X 0,Y 277.235,Z 496.776,A -85,B 0,C 180,E1 -17383.935,E2 -17383.935} C_VEL
LIN {X 0,Y 278.348,Z 487.122,A -85,B 0,C 180,E1 -17386.125,E2 -17386.125} C_VEL
LIN {X 0,Y 279.652,Z 477.114,A -85,B 0,C 180,E1 -17387.93,E2 -17387.93} C_VEL
LIN {X 0,Y 279.713,Z 465.538,A -85,B 0,C 180,E1 -17389.636,E2 -17389.636} C_VEL
LIN {X 0,Y 279.321,Z 454.055,A -85,B 0,C 180,E1 -17391.011,E2 -17391.011} C_VEL
LIN {X 0,Y 278.736,Z 441.283,A -85,B 0,C 180,E1 -17392.222,E2 -17392.222} C_VEL
LIN {X 0,Y 277.785,Z 427.731,A -85,B 0,C 180,E1 -17393.211,E2 -17393.211} C_VEL
LIN {X 0,Y 276.915,Z 416.699,A -85,B 0,C 180,E1 -17393.858,E2 -17393.858} C_VEL
LIN {X 0,Y 277.45,Z 410.735,A -85,B 0,C 180,E1 -17396.313,E2 -17396.313} C_VEL
LIN {X 0,Y 278.759,Z 399.95,A -85,B 0,C 180,E1 -17400.996,E2 -17400.996} C_VEL
LIN {X 0,Y 280.298,Z 390.366,A -85,B 0,C 180,E1 -17405.217,E2 -17405.217} C_VEL
LIN {X 0,Y 281.348,Z 384.718,A -85,B 0,C 180,E1 -17407.733,E2 -17407.733} C_VEL
LIN {X 0,Y 281.264,Z 381.463,A -85,B 0,C 180,E1 -17409.231,E2 -17409.231} C_VEL
LIN {X 0,Y 279.662,Z 373.329,A -85,B 0,C 180,E1 -17413.216,E2 -17413.216} C_VEL
LIN {X 0,Y 278.183,Z 365.748,A -85,B 0,C 180,E1 -17417.108,E2 -17417.108} C_VEL
LIN {X 0,Y 277.272,Z 360.992,A -85,B 0,C 180,E1 -17419.79,E2 -17419.79} C_VEL
LIN {X 0,Y 277.275,Z 360.945,A -85,B 0,C 180,E1 -17424.34,E2 -17424.34} C_VEL
LIN {X 0,Y 277.24,Z 360.949,A -85,B 0,C 180,E1 -17427.836,E2 -17427.836} C_VEL
LIN {X 0,Y 277.284,Z 360.946,A -85,B 0,C 180,E1 -17431.212,E2 -17431.212} C_VEL
LIN {X 0,Y 277.302,Z 360.941,A -85,B 0,C 180,E1 -17434.478,E2 -17434.478} C_VEL
LIN {X 0,Y 277.26,Z 360.945,A -85,B 0,C 180,E1 -17437.653,E2 -17437.653} C_VEL
LIN {X 0,Y 277.311,Z 360.941,A -85,B 0,C 180,E1 -17440.764,E2 -17440.764} C_VEL
LIN {X 0,Y 277.403,Z 360.928,A -85,B 0,C 180,E1 -17445.324,E2 -17445.324} C_VEL
LIN {X 0,Y 277.448,Z 360.922,A -85,B 0,C 180,E1 -17449.786,E2 -17449.786} C_VEL
LIN {X 0,Y 277.615,Z 360.905,A -85,B 0,C 180,E1 -17452.728,E2 -17452.728} C_VEL
LIN {X 0,Y 277.813,Z 360.878,A -85,B 0,C 180,E1 -17458.55,E2 -17458.55} C_VEL
LIN {X 0,Y 277.813,Z 360.877,A -85,B 0,C 180,E1 -17461.45,E2 -17461.45} C_VEL
LIN {X 0,Y 277.642,Z 360.899,A -85,B 0,C 180,E1 -17467.271,E2 -17467.271} C_VEL
LIN {X 0,Y 277.5,Z 360.917,A -85,B 0,C 180,E1 -17470.212,E2 -17470.212} C_VEL
LIN {X 0,Y 277.422,Z 360.93,A -85,B 0,C 180,E1 -17474.675,E2 -17474.675} C_VEL
LIN {X 0,Y 277.339,Z 360.936,A -85,B 0,C 180,E1 -17479.234,E2 -17479.234} C_VEL
LIN {X 0,Y 277.313,Z 360.941,A -85,B 0,C 180,E1 -17484.171,E2 -17484.171} C_VEL
LIN {X 0,Y 277.321,Z 360.938,A -85,B 0,C 180,E1 -17487.506,E2 -17487.506} C_VEL
LIN {X 0,Y 277.267,Z 360.948,A -85,B 0,C 180,E1 -17490.482,E2 -17490.482} C_VEL
LIN {X 0,Y 277.25,Z 360.949,A -85,B 0,C 180,E1 -17493.895,E2 -17493.895} C_VEL
LIN {X 0,Y 277.28,Z 360.942,A -85,B 0,C 180,E1 -17497.467,E2 -17497.467} C_VEL
LIN {X 0,Y 277.236,Z 360.949,A -85,B 0,C 180,E1 -17501.232,E2 -17501.232} C_VEL
LIN {X 0,Y 277.202,Z 360.952,A -85,B 0,C 180,E1 -17505.226,E2 -17505.226} C_VEL
LIN {X 0,Y 277.22,Z 360.951,A -85,B 0,C 180,E1 -17509.513,E2 -17509.513} C_VEL
LIN {X 0,Y 277.272,Z 360.945,A -85,B 0,C 180,E1 -17512.532,E2 -17512.532} C_VEL
LIN {X 0,Y 277.246,Z 360.951,A -85,B 0,C 180,E1 -17516.105,E2 -17516.105} C_VEL
LIN {X 0,Y 277.261,Z 360.947,A -85,B 0,C 180,E1 -17519.539,E2 -17519.539} C_VEL
LIN {X 0,Y 277.36,Z 360.932,A -85,B 0,C 180,E1 -17522.865,E2 -17522.865} C_VEL
LIN {X 0,Y 277.329,Z 360.94,A -85,B 0,C 180,E1 -17526.08,E2 -17526.08} C_VEL
LIN {X 0,Y 277.346,Z 360.934,A -85,B 0,C 180,E1 -17530.767,E2 -17530.767} C_VEL
LIN {X 0,Y 277.436,Z 360.925,A -85,B 0,C 180,E1 -17535.326,E2 -17535.326} C_VEL
LIN {X 0,Y 277.508,Z 360.918,A -85,B 0,C 180,E1 -17539.789,E2 -17539.789} C_VEL
LIN {X 0,Y 277.656,Z 360.896,A -85,B 0,C 180,E1 -17542.729,E2 -17542.729} C_VEL
LIN {X 0,Y 277.827,Z 360.875,A -85,B 0,C 180,E1 -17548.551,E2 -17548.551} C_VEL
LIN {X 0,Y 277.824,Z 360.88,A -85,B 0,C 180,E1 -17551.45,E2 -17551.45} C_VEL
LIN {X 0,Y 277.646,Z 360.9,A -85,B 0,C 180,E1 -17557.271,E2 -17557.271} C_VEL
LIN {X 0,Y 277.508,Z 360.915,A -85,B 0,C 180,E1 -17560.211,E2 -17560.211} C_VEL
LIN {X 0,Y 277.436,Z 360.924,A -85,B 0,C 180,E1 -17564.674,E2 -17564.674} C_VEL
LIN {X 0,Y 277.346,Z 360.94,A -85,B 0,C 180,E1 -17569.233,E2 -17569.233} C_VEL
LIN {X 0,Y 277.319,Z 360.938,A -85,B 0,C 180,E1 -17574.17,E2 -17574.17} C_VEL
LIN {X 0,Y 277.322,Z 360.94,A -85,B 0,C 180,E1 -17577.503,E2 -17577.503} C_VEL
LIN {X 0,Y 277.271,Z 360.946,A -85,B 0,C 180,E1 -17580.481,E2 -17580.481} C_VEL
LIN {X 0,Y 277.253,Z 360.948,A -85,B 0,C 180,E1 -17583.894,E2 -17583.894} C_VEL
LIN {X 0,Y 277.29,Z 360.946,A -85,B 0,C 180,E1 -17587.465,E2 -17587.465} C_VEL
LIN {X 0,Y 277.343,Z 361.088,A -85,B 0,C 180,E1 -17589.678,E2 -17589.678} C_VEL
LIN {X 0,Y 277.59,Z 362.159,A -85,B 0,C 180,E1 -17589.932,E2 -17589.932} C_VEL
LIN {X 0,Y 281.183,Z 374.401,A -85,B 0,C 180,E1 -17591.334,E2 -17591.334} C_VEL
LIN {X 0,Y 284.048,Z 385.742,A -85,B 0,C 180,E1 -17592.874,E2 -17592.874} C_VEL
LIN {X 0,Y 282.922,Z 396.791,A -85,B 0,C 180,E1 -17594.448,E2 -17594.448} C_VEL
LIN {X 0,Y 281.759,Z 406.35,A -85,B 0,C 180,E1 -17596.112,E2 -17596.112} C_VEL
LIN {X 0,Y 280.554,Z 416.071,A -85,B 0,C 180,E1 -17598.206,E2 -17598.206} C_VEL
LIN {X 0,Y 279.662,Z 423.44,A -85,B 0,C 180,E1 -17600.147,E2 -17600.147} C_VEL
LIN {X 0,Y 278.832,Z 430.375,A -85,B 0,C 180,E1 -17602.387,E2 -17602.387} C_VEL
LIN {X 0,Y 278.27,Z 435.567,A -85,B 0,C 180,E1 -17604.487,E2 -17604.487} C_VEL
LIN {X 0,Y 277.839,Z 440.749,A -85,B 0,C 180,E1 -17607.236,E2 -17607.236} C_VEL
LIN {X 0,Y 277.64,Z 443.916,A -85,B 0,C 180,E1 -17609.584,E2 -17609.584} C_VEL
LIN {X 0,Y 277.72,Z 446.221,A -85,B 0,C 180,E1 -17612.337,E2 -17612.337} C_VEL
LIN {X 0,Y 278.272,Z 447.106,A -85,B 0,C 180,E1 -17615.393,E2 -17615.393} C_VEL
LIN {X 0,Y 279.342,Z 446.121,A -85,B 0,C 180,E1 -17618.57,E2 -17618.57} C_VEL
LIN {X 0,Y 280.436,Z 444.1,A -85,B 0,C 180,E1 -17620.986,E2 -17620.986} C_VEL
LIN {X 0,Y 281.803,Z 440.96,A -85,B 0,C 180,E1 -17623.333,E2 -17623.333} C_VEL
LIN {X 0,Y 283.484,Z 436.571,A -85,B 0,C 180,E1 -17625.646,E2 -17625.646} C_VEL
LIN {X 0,Y 285.513,Z 430.876,A -85,B 0,C 180,E1 -17627.923,E2 -17627.923} C_VEL
LIN {X 0,Y 287.81,Z 423.703,A -85,B 0,C 180,E1 -17630.158,E2 -17630.158} C_VEL
LIN {X 0,Y 290.238,Z 415.084,A -85,B 0,C 180,E1 -17632.25,E2 -17632.25} C_VEL
LIN {X 0,Y 292.681,Z 405.282,A -85,B 0,C 180,E1 -17634.143,E2 -17634.143} C_VEL
LIN {X 0,Y 293.521,Z 401.352,A -85,B 0,C 180,E1 -17634.794,E2 -17634.794} C_VEL
LIN {X 0,Y 293.298,Z 398.48,A -85,B 0,C 180,E1 -17635.369,E2 -17635.369} C_VEL
LIN {X 0,Y 291.571,Z 391.304,A -85,B 0,C 180,E1 -17636.891,E2 -17636.891} C_VEL
LIN {X 0,Y 287.675,Z 380.503,A -85,B 0,C 180,E1 -17639.158,E2 -17639.158} C_VEL
LIN {X 0,Y 283.367,Z 371.125,A -85,B 0,C 180,E1 -17641.103,E2 -17641.103} C_VEL
LIN {X 0,Y 280.235,Z 365.497,A -85,B 0,C 180,E1 -17642.335,E2 -17642.335} C_VEL
LIN {X 0,Y 278.072,Z 362.593,A -85,B 0,C 180,E1 -17643.079,E2 -17643.079} C_VEL
LIN {X 0,Y 277.628,Z 361.254,A -85,B 0,C 180,E1 -17643.447,E2 -17643.447} C_VEL
LIN {X 0,Y 277.481,Z 360.922,A -85,B 0,C 180,E1 -17643.994,E2 -17643.994} C_VEL
LIN {X 0,Y 277.62,Z 360.905,A -85,B 0,C 180,E1 -17647.272,E2 -17647.272} C_VEL
LIN {X 0,Y 277.557,Z 360.912,A -85,B 0,C 180,E1 -17648.963,E2 -17648.963} C_VEL
LIN {X 0,Y 276.868,Z 361.004,A -85,B 0,C 180,E1 -17650.172,E2 -17650.172} C_VEL
LIN {X 0,Y 273.98,Z 361.364,A -85,B 0,C 180,E1 -17652.141,E2 -17652.141} C_VEL
LIN {X 0,Y 271.521,Z 361.665,A -85,B 0,C 180,E1 -17653.74,E2 -17653.74} C_VEL
LIN {X 0,Y 270.442,Z 361.798,A -85,B 0,C 180,E1 -17654.981,E2 -17654.981} C_VEL
LIN {X 0,Y 270.34,Z 361.81,A -85,B 0,C 180,E1 -17655.402,E2 -17655.402} C_VEL
LIN {X 0,Y 270.252,Z 361.818,A -85,B 0,C 180,E1 -17659.759,E2 -17659.759} C_VEL
LIN {X 0,Y 270.232,Z 361.821,A -85,B 0,C 180,E1 -17664.59,E2 -17664.59} C_VEL
LIN {X 0,Y 270.305,Z 361.877,A -85,B 0,C 180,E1 -17667.458,E2 -17667.458} C_VEL
LIN {X 0,Y 270.611,Z 363.238,A -85,B 0,C 180,E1 -17669.567,E2 -17669.567} C_VEL
LIN {X 0,Y 271.289,Z 366.838,A -85,B 0,C 180,E1 -17674.007,E2 -17674.007} C_VEL
LIN {X 0,Y 271.88,Z 369.476,A -85,B 0,C 180,E1 -17676.744,E2 -17676.744} C_VEL
LIN {X 0,Y 272.695,Z 373.253,A -85,B 0,C 180,E1 -17680.114,E2 -17680.114} C_VEL
LIN {X 0,Y 273.765,Z 378.331,A -85,B 0,C 180,E1 -17684.045,E2 -17684.045} C_VEL
LIN {X 0,Y 274.973,Z 384.835,A -85,B 0,C 180,E1 -17688.355,E2 -17688.355} C_VEL
LIN {X 0,Y 275.456,Z 388.18,A -85,B 0,C 180,E1 -17690.369,E2 -17690.369} C_VEL
LIN {X 0,Y 275.404,Z 389.874,A -85,B 0,C 180,E1 -17691.303,E2 -17691.303} C_VEL
LIN {X 0,Y 273.408,Z 398.405,A -85,B 0,C 180,E1 -17695.563,E2 -17695.563} C_VEL
LIN {X 0,Y 272.833,Z 401.572,A -85,B 0,C 180,E1 -17696.978,E2 -17696.978} C_VEL
LIN {X 0,Y 273.327,Z 404.604,A -85,B 0,C 180,E1 -17697.397,E2 -17697.397} C_VEL
LIN {X 0,Y 274.492,Z 408.519,A -85,B 0,C 180,E1 -17697.907,E2 -17697.907} C_VEL
LIN {X 0,Y 276.675,Z 417.585,A -85,B 0,C 180,E1 -17699.029,E2 -17699.029} C_VEL
LIN {X 0,Y 278.778,Z 430.048,A -85,B 0,C 180,E1 -17700.582,E2 -17700.582} C_VEL
LIN {X 0,Y 279.853,Z 442.203,A -85,B 0,C 180,E1 -17702.131,E2 -17702.131} C_VEL
LIN {X 0,Y 279.924,Z 453.927,A -85,B 0,C 180,E1 -17703.737,E2 -17703.737} C_VEL
LIN {X 0,Y 278.882,Z 465.682,A -85,B 0,C 180,E1 -17705.514,E2 -17705.514} C_VEL
LIN {X 0,Y 277.284,Z 475.807,A -85,B 0,C 180,E1 -17707.262,E2 -17707.262} C_VEL
LIN {X 0,Y 275.643,Z 484.744,A -85,B 0,C 180,E1 -17709.087,E2 -17709.087} C_VEL
LIN {X 0,Y 273.252,Z 493.744,A -85,B 0,C 180,E1 -17711.247,E2 -17711.247} C_VEL
LIN {X 0,Y 271.2,Z 501.867,A -85,B 0,C 180,E1 -17713.677,E2 -17713.677} C_VEL
LIN {X 0,Y 270.604,Z 505.427,A -85,B 0,C 180,E1 -17714.947,E2 -17714.947} C_VEL
LIN {X 0,Y 269.544,Z 510.802,A -85,B 0,C 180,E1 -17717.196,E2 -17717.196} C_VEL
LIN {X 0,Y 268.984,Z 515.111,A -85,B 0,C 180,E1 -17719.462,E2 -17719.462} C_VEL
LIN {X 0,Y 268.982,Z 519.382,A -85,B 0,C 180,E1 -17722.494,E2 -17722.494} C_VEL
LIN {X 0,Y 269.47,Z 521.933,A -85,B 0,C 180,E1 -17725.513,E2 -17725.513} C_VEL
LIN {X 0,Y 270.211,Z 522.872,A -85,B 0,C 180,E1 -17728.51,E2 -17728.51} C_VEL
LIN {X 0,Y 270.563,Z 522.665,A -85,B 0,C 180,E1 -17730,E2 -17730} C_VEL
LIN {X 0,Y 270.272,Z 521.923,A -85,B 0,C 180,E1 -17731.49,E2 -17731.49} C_VEL
LIN {X 0,Y 269.938,Z 520.74,A -85,B 0,C 180,E1 -17732.985,E2 -17732.985} C_VEL
LIN {X 0,Y 269.72,Z 518.105,A -85,B 0,C 180,E1 -17735.232,E2 -17735.232} C_VEL
LIN {X 0,Y 269.413,Z 514.169,A -85,B 0,C 180,E1 -17737.571,E2 -17737.571} C_VEL
LIN {X 0,Y 269.286,Z 509.305,A -85,B 0,C 180,E1 -17739.767,E2 -17739.767} C_VEL
LIN {X 0,Y 269.607,Z 502.955,A -85,B 0,C 180,E1 -17742.037,E2 -17742.037} C_VEL
LIN {X 0,Y 270.273,Z 495.01,A -85,B 0,C 180,E1 -17744.302,E2 -17744.302} C_VEL
LIN {X 0,Y 271.271,Z 486.965,A -85,B 0,C 180,E1 -17746.171,E2 -17746.171} C_VEL
LIN {X 0,Y 272.57,Z 477.207,A -85,B 0,C 180,E1 -17748.023,E2 -17748.023} C_VEL
LIN {X 0,Y 272.652,Z 465.854,A -85,B 0,C 180,E1 -17749.774,E2 -17749.774} C_VEL
LIN {X 0,Y 272.303,Z 454.741,A -85,B 0,C 180,E1 -17751.182,E2 -17751.182} C_VEL
LIN {X 0,Y 271.772,Z 441.915,A -85,B 0,C 180,E1 -17752.475,E2 -17752.475} C_VEL
LIN {X 0,Y 270.838,Z 427.697,A -85,B 0,C 180,E1 -17753.566,E2 -17753.566} C_VEL
LIN {X 0,Y 269.904,Z 415.614,A -85,B 0,C 180,E1 -17754.305,E2 -17754.305} C_VEL
LIN {X 0,Y 270.978,Z 405.568,A -85,B 0,C 180,E1 -17758.714,E2 -17758.714} C_VEL
LIN {X 0,Y 272.305,Z 396.459,A -85,B 0,C 180,E1 -17762.819,E2 -17762.819} C_VEL
LIN {X 0,Y 274.064,Z 386.486,A -85,B 0,C 180,E1 -17767.349,E2 -17767.349} C_VEL
LIN {X 0,Y 274.355,Z 383.38,A -85,B 0,C 180,E1 -17768.791,E2 -17768.791} C_VEL
LIN {X 0,Y 272.805,Z 375.179,A -85,B 0,C 180,E1 -17772.887,E2 -17772.887} C_VEL
LIN {X 0,Y 271.272,Z 367.26,A -85,B 0,C 180,E1 -17777.043,E2 -17777.043} C_VEL
LIN {X 0,Y 270.23,Z 361.894,A -85,B 0,C 180,E1 -17780.055,E2 -17780.055} C_VEL
LIN {X 0,Y 270.217,Z 361.826,A -85,B 0,C 180,E1 -17783.731,E2 -17783.731} C_VEL
LIN {X 0,Y 270.198,Z 361.828,A -85,B 0,C 180,E1 -17786.892,E2 -17786.892} C_VEL
LIN {X 0,Y 270.224,Z 361.822,A -85,B 0,C 180,E1 -17790.386,E2 -17790.386} C_VEL
LIN {X 0,Y 270.254,Z 361.819,A -85,B 0,C 180,E1 -17793.763,E2 -17793.763} C_VEL
LIN {X 0,Y 270.203,Z 361.828,A -85,B 0,C 180,E1 -17797.036,E2 -17797.036} C_VEL
LIN {X 0,Y 270.252,Z 361.819,A -85,B 0,C 180,E1 -17800.241,E2 -17800.241} C_VEL
LIN {X 0,Y 270.362,Z 361.808,A -85,B 0,C 180,E1 -17804.933,E2 -17804.933} C_VEL
LIN {X 0,Y 270.4,Z 361.8,A -85,B 0,C 180,E1 -17809.517,E2 -17809.517} C_VEL
LIN {X 0,Y 270.573,Z 361.781,A -85,B 0,C 180,E1 -17812.538,E2 -17812.538} C_VEL
LIN {X 0,Y 270.779,Z 361.754,A -85,B 0,C 180,E1 -17818.513,E2 -17818.513} C_VEL
LIN {X 0,Y 270.779,Z 361.753,A -85,B 0,C 180,E1 -17821.487,E2 -17821.487} C_VEL
LIN {X 0,Y 270.601,Z 361.775,A -85,B 0,C 180,E1 -17827.461,E2 -17827.461} C_VEL
LIN {X 0,Y 270.435,Z 361.799,A -85,B 0,C 180,E1 -17830.481,E2 -17830.481} C_VEL
LIN {X 0,Y 270.39,Z 361.802,A -85,B 0,C 180,E1 -17835.065,E2 -17835.065} C_VEL
LIN {X 0,Y 270.296,Z 361.813,A -85,B 0,C 180,E1 -17839.756,E2 -17839.756} C_VEL
LIN {X 0,Y 270.269,Z 361.82,A -85,B 0,C 180,E1 -17844.586,E2 -17844.586} C_VEL
LIN {X 0,Y 270.267,Z 361.818,A -85,B 0,C 180,E1 -17847.909,E2 -17847.909} C_VEL
LIN {X 0,Y 270.18,Z 361.827,A -85,B 0,C 180,E1 -17851.349,E2 -17851.349} C_VEL
LIN {X 0,Y 270.211,Z 361.825,A -85,B 0,C 180,E1 -17854.904,E2 -17854.904} C_VEL
LIN {X 0,Y 270.219,Z 361.823,A -85,B 0,C 180,E1 -17858.718,E2 -17858.718} C_VEL
LIN {X 0,Y 270.188,Z 361.829,A -85,B 0,C 180,E1 -17862.555,E2 -17862.555} C_VEL
LIN {X 0,Y 270.163,Z 361.829,A -85,B 0,C 180,E1 -17866.752,E2 -17866.752} C_VEL
LIN {X 0,Y 270.172,Z 361.829,A -85,B 0,C 180,E1 -17869.435,E2 -17869.435} C_VEL
LIN {X 0,Y 270.242,Z 361.822,A -85,B 0,C 180,E1 -17873.726,E2 -17873.726} C_VEL
LIN {X 0,Y 270.203,Z 361.825,A -85,B 0,C 180,E1 -17876.893,E2 -17876.893} C_VEL
LIN {X 0,Y 270.235,Z 361.822,A -85,B 0,C 180,E1 -17880.388,E2 -17880.388} C_VEL
LIN {X 0,Y 270.265,Z 361.819,A -85,B 0,C 180,E1 -17883.765,E2 -17883.765} C_VEL
LIN {X 0,Y 270.233,Z 361.821,A -85,B 0,C 180,E1 -17887.039,E2 -17887.039} C_VEL
LIN {X 0,Y 270.302,Z 361.813,A -85,B 0,C 180,E1 -17890.245,E2 -17890.245} C_VEL
LIN {X 0,Y 270.404,Z 361.8,A -85,B 0,C 180,E1 -17894.936,E2 -17894.936} C_VEL
LIN {X 0,Y 270.443,Z 361.797,A -85,B 0,C 180,E1 -17899.519,E2 -17899.519} C_VEL
LIN {X 0,Y 270.614,Z 361.774,A -85,B 0,C 180,E1 -17902.539,E2 -17902.539} C_VEL
LIN {X 0,Y 270.792,Z 361.751,A -85,B 0,C 180,E1 -17908.513,E2 -17908.513} C_VEL
LIN {X 0,Y 270.79,Z 361.756,A -85,B 0,C 180,E1 -17911.487,E2 -17911.487} C_VEL
LIN {X 0,Y 270.604,Z 361.779,A -85,B 0,C 180,E1 -17917.461,E2 -17917.461} C_VEL
LIN {X 0,Y 270.443,Z 361.795,A -85,B 0,C 180,E1 -17920.481,E2 -17920.481} C_VEL
LIN {X 0,Y 270.404,Z 361.803,A -85,B 0,C 180,E1 -17925.064,E2 -17925.064} C_VEL
LIN {X 0,Y 270.302,Z 361.814,A -85,B 0,C 180,E1 -17929.755,E2 -17929.755} C_VEL
LIN {X 0,Y 270.274,Z 361.817,A -85,B 0,C 180,E1 -17934.585,E2 -17934.585} C_VEL
LIN {X 0,Y 270.269,Z 361.817,A -85,B 0,C 180,E1 -17937.908,E2 -17937.908} C_VEL
LIN {X 0,Y 270.183,Z 361.831,A -85,B 0,C 180,E1 -17941.347,E2 -17941.347} C_VEL
LIN {X 0,Y 270.215,Z 361.828,A -85,B 0,C 180,E1 -17944.903,E2 -17944.903} C_VEL
LIN {X 0,Y 270.264,Z 361.868,A -85,B 0,C 180,E1 -17949.213,E2 -17949.213} C_VEL
LIN {X 0,Y 270.484,Z 362.928,A -85,B 0,C 180,E1 -17949.535,E2 -17949.535} C_VEL
LIN {X 0,Y 274.28,Z 375.779,A -85,B 0,C 180,E1 -17951.046,E2 -17951.046} C_VEL
LIN {X 0,Y 276.85,Z 385.547,A -85,B 0,C 180,E1 -17952.406,E2 -17952.406} C_VEL
LIN {X 0,Y 277.107,Z 387.2,A -85,B 0,C 180,E1 -17952.65,E2 -17952.65} C_VEL
LIN {X 0,Y 275.92,Z 398.213,A -85,B 0,C 180,E1 -17954.266,E2 -17954.266} C_VEL
LIN {X 0,Y 274.736,Z 407.79,A -85,B 0,C 180,E1 -17955.996,E2 -17955.996} C_VEL
LIN {X 0,Y 273.477,Z 417.612,A -85,B 0,C 180,E1 -17958.18,E2 -17958.18} C_VEL
LIN {X 0,Y 272.545,Z 425.54,A -85,B 0,C 180,E1 -17960.366,E2 -17960.366} C_VEL
LIN {X 0,Y 271.595,Z 433.139,A -85,B 0,C 180,E1 -17963.014,E2 -17963.014} C_VEL
LIN {X 0,Y 271.112,Z 438.121,A -85,B 0,C 180,E1 -17965.229,E2 -17965.229} C_VEL
LIN {X 0,Y 270.712,Z 442.604,A -85,B 0,C 180,E1 -17967.845,E2 -17967.845} C_VEL
LIN {X 0,Y 270.601,Z 445.675,A -85,B 0,C 180,E1 -17970.431,E2 -17970.431} C_VEL
LIN {X 0,Y 270.679,Z 447.053,A -85,B 0,C 180,E1 -17972.137,E2 -17972.137} C_VEL
LIN {X 0,Y 271.176,Z 448.143,A -85,B 0,C 180,E1 -17975.103,E2 -17975.103} C_VEL
LIN {X 0,Y 271.798,Z 447.992,A -85,B 0,C 180,E1 -17977.178,E2 -17977.178} C_VEL
LIN {X 0,Y 272.433,Z 447.297,A -85,B 0,C 180,E1 -17978.829,E2 -17978.829} C_VEL
LIN {X 0,Y 273.174,Z 446.152,A -85,B 0,C 180,E1 -17980.461,E2 -17980.461} C_VEL
LIN {X 0,Y 274.518,Z 443.47,A -85,B 0,C 180,E1 -17982.878,E2 -17982.878} C_VEL
LIN {X 0,Y 276.216,Z 439.617,A -85,B 0,C 180,E1 -17985.26,E2 -17985.26} C_VEL
LIN {X 0,Y 278.264,Z 434.483,A -85,B 0,C 180,E1 -17987.603,E2 -17987.603} C_VEL
LIN {X 0,Y 280.544,Z 427.973,A -85,B 0,C 180,E1 -17989.9,E2 -17989.9} C_VEL
LIN {X 0,Y 283.094,Z 419.87,A -85,B 0,C 180,E1 -17992.109,E2 -17992.109} C_VEL
LIN {X 0,Y 285.523,Z 411.282,A -85,B 0,C 180,E1 -17993.995,E2 -17993.995} C_VEL
LIN {X 0,Y 287.487,Z 403.244,A -85,B 0,C 180,E1 -17995.443,E2 -17995.443} C_VEL
LIN {X 0,Y 286.232,Z 396.33,A -85,B 0,C 180,E1 -17996.981,E2 -17996.981} C_VEL
LIN {X 0,Y 282.888,Z 386.191,A -85,B 0,C 180,E1 -17999.288,E2 -17999.288} C_VEL
LIN {X 0,Y 279.552,Z 377.823,A -85,B 0,C 180,E1 -18001.118,E2 -18001.118} C_VEL
LIN {X 0,Y 276.352,Z 371.743,A -85,B 0,C 180,E1 -18002.551,E2 -18002.551} C_VEL
LIN {X 0,Y 273.082,Z 366.474,A -85,B 0,C 180,E1 -18003.873,E2 -18003.873} C_VEL
LIN {X 0,Y 271.466,Z 364.719,A -85,B 0,C 180,E1 -18004.455,E2 -18004.455} C_VEL
LIN {X 0,Y 270.529,Z 362.291,A -85,B 0,C 180,E1 -18005.03,E2 -18005.03} C_VEL
LIN {X 0,Y 270.481,Z 361.799,A -85,B 0,C 180,E1 -18005.592,E2 -18005.592} C_VEL
LIN {X 0,Y 270.521,Z 361.789,A -85,B 0,C 180,E1 -18008.968,E2 -18008.968} C_VEL
LIN {X 0,Y 270.34,Z 361.81,A -85,B 0,C 180,E1 -18013.531,E2 -18013.531} C_VEL
LIN {X 0,Y 270.34,Z 361.81,A -85,B 0,C 180,E1 -18015.402,E2 -18015.402} C_VEL
LIN {X 0,Y 269.634,Z 361.901,A -85,B 0,C 180,E1 -18016.644,E2 -18016.644} C_VEL
LIN {X 0,Y 266.754,Z 362.268,A -85,B 0,C 180,E1 -18018.667,E2 -18018.667} C_VEL
LIN {X 0,Y 264.311,Z 362.572,A -85,B 0,C 180,E1 -18020.312,E2 -18020.312} C_VEL
LIN {X 0,Y 263.236,Z 362.698,A -85,B 0,C 180,E1 -18021.587,E2 -18021.587} C_VEL
LIN {X 0,Y 263.134,Z 362.706,A -85,B 0,C 180,E1 -18022.02,E2 -18022.02} C_VEL
LIN {X 0,Y 263.195,Z 362.761,A -85,B 0,C 180,E1 -18024.788,E2 -18024.788} C_VEL
LIN {X 0,Y 263.69,Z 364.791,A -85,B 0,C 180,E1 -18028.417,E2 -18028.417} C_VEL
LIN {X 0,Y 264.212,Z 367.498,A -85,B 0,C 180,E1 -18032.141,E2 -18032.141} C_VEL
LIN {X 0,Y 264.909,Z 370.668,A -85,B 0,C 180,E1 -18035.708,E2 -18035.708} C_VEL
LIN {X 0,Y 265.897,Z 375.182,A -85,B 0,C 180,E1 -18039.96,E2 -18039.96} C_VEL
LIN {X 0,Y 266.947,Z 380.271,A -85,B 0,C 180,E1 -18043.984,E2 -18043.984} C_VEL
LIN {X 0,Y 268.054,Z 386.389,A -85,B 0,C 180,E1 -18048.178,E2 -18048.178} C_VEL
LIN {X 0,Y 268.555,Z 389.77,A -85,B 0,C 180,E1 -18050.28,E2 -18050.28} C_VEL
LIN {X 0,Y 268.167,Z 392.619,A -85,B 0,C 180,E1 -18051.835,E2 -18051.835} C_VEL
LIN {X 0,Y 266.464,Z 399.904,A -85,B 0,C 180,E1 -18055.454,E2 -18055.454} C_VEL
LIN {X 0,Y 267.364,Z 404.152,A -85,B 0,C 180,E1 -18056.076,E2 -18056.076} C_VEL
LIN {X 0,Y 269.703,Z 413.111,A -85,B 0,C 180,E1 -18057.288,E2 -18057.288} C_VEL
LIN {X 0,Y 272.179,Z 426.078,A -85,B 0,C 180,E1 -18059.033,E2 -18059.033} C_VEL
LIN {X 0,Y 273.403,Z 437.629,A -85,B 0,C 180,E1 -18060.587,E2 -18060.587} C_VEL
LIN {X 0,Y 273.74,Z 450.887,A -85,B 0,C 180,E1 -18062.476,E2 -18062.476} C_VEL
LIN {X 0,Y 273.115,Z 461.181,A -85,B 0,C 180,E1 -18064.059,E2 -18064.059} C_VEL
LIN {X 0,Y 271.502,Z 472.15,A -85,B 0,C 180,E1 -18065.94,E2 -18065.94} C_VEL
LIN {X 0,Y 269.353,Z 483.081,A -85,B 0,C 180,E1 -18068.173,E2 -18068.173} C_VEL
LIN {X 0,Y 266.891,Z 492.162,A -85,B 0,C 180,E1 -18070.383,E2 -18070.383} C_VEL
LIN {X 0,Y 264.854,Z 499.66,A -85,B 0,C 180,E1 -18072.632,E2 -18072.632} C_VEL
LIN {X 0,Y 263.219,Z 506.756,A -85,B 0,C 180,E1 -18075.307,E2 -18075.307} C_VEL
LIN {X 0,Y 262.273,Z 511.656,A -85,B 0,C 180,E1 -18077.622,E2 -18077.622} C_VEL
LIN {X 0,Y 261.819,Z 516.643,A -85,B 0,C 180,E1 -18080.732,E2 -18080.732} C_VEL
LIN {X 0,Y 262.091,Z 519.908,A -85,B 0,C 180,E1 -18083.843,E2 -18083.843} C_VEL
LIN {X 0,Y 262.39,Z 520.947,A -85,B 0,C 180,E1 -18085.391,E2 -18085.391} C_VEL
LIN {X 0,Y 262.672,Z 521.572,A -85,B 0,C 180,E1 -18086.933,E2 -18086.933} C_VEL
LIN {X 0,Y 263.169,Z 521.769,A -85,B 0,C 180,E1 -18088.47,E2 -18088.47} C_VEL
LIN {X 0,Y 263.54,Z 521.516,A -85,B 0,C 180,E1 -18090,E2 -18090} C_VEL
LIN {X 0,Y 263.239,Z 520.732,A -85,B 0,C 180,E1 -18091.53,E2 -18091.53} C_VEL
LIN {X 0,Y 262.904,Z 519.499,A -85,B 0,C 180,E1 -18093.065,E2 -18093.065} C_VEL
LIN {X 0,Y 262.681,Z 516.77,A -85,B 0,C 180,E1 -18095.373,E2 -18095.373} C_VEL
LIN {X 0,Y 262.355,Z 512.866,A -85,B 0,C 180,E1 -18097.697,E2 -18097.697} C_VEL
LIN {X 0,Y 262.26,Z 507.727,A -85,B 0,C 180,E1 -18100.031,E2 -18100.031} C_VEL
LIN {X 0,Y 262.604,Z 501.239,A -85,B 0,C 180,E1 -18102.363,E2 -18102.363} C_VEL
LIN {X 0,Y 263.356,Z 493.174,A -85,B 0,C 180,E1 -18104.686,E2 -18104.686} C_VEL
LIN {X 0,Y 264.425,Z 484.51,A -85,B 0,C 180,E1 -18106.7,E2 -18106.7} C_VEL
LIN {X 0,Y 265.608,Z 476.186,A -85,B 0,C 180,E1 -18108.293,E2 -18108.293} C_VEL
LIN {X 0,Y 265.591,Z 464.616,A -85,B 0,C 180,E1 -18110.12,E2 -18110.12} C_VEL
LIN {X 0,Y 265.229,Z 453.399,A -85,B 0,C 180,E1 -18111.571,E2 -18111.571} C_VEL
LIN {X 0,Y 264.716,Z 441.021,A -85,B 0,C 180,E1 -18112.846,E2 -18112.846} C_VEL
LIN {X 0,Y 263.827,Z 426.968,A -85,B 0,C 180,E1 -18113.961,E2 -18113.961} C_VEL
LIN {X 0,Y 262.873,Z 414.872,A -85,B 0,C 180,E1 -18114.712,E2 -18114.712} C_VEL
LIN {X 0,Y 263.202,Z 411.493,A -85,B 0,C 180,E1 -18116.14,E2 -18116.14} C_VEL
LIN {X 0,Y 264.362,Z 402.388,A -85,B 0,C 180,E1 -18120.338,E2 -18120.338} C_VEL
LIN {X 0,Y 265.999,Z 392.338,A -85,B 0,C 180,E1 -18125.009,E2 -18125.009} C_VEL
LIN {X 0,Y 267.198,Z 386.212,A -85,B 0,C 180,E1 -18127.9,E2 -18127.9} C_VEL
LIN {X 0,Y 267.064,Z 382.608,A -85,B 0,C 180,E1 -18129.662,E2 -18129.662} C_VEL
LIN {X 0,Y 265.275,Z 373.625,A -85,B 0,C 180,E1 -18134.33,E2 -18134.33} C_VEL
LIN {X 0,Y 263.834,Z 366.473,A -85,B 0,C 180,E1 -18138.245,E2 -18138.245} C_VEL
LIN {X 0,Y 263.165,Z 362.768,A -85,B 0,C 180,E1 -18140.421,E2 -18140.421} C_VEL
LIN {X 0,Y 263.155,Z 362.705,A -85,B 0,C 180,E1 -18144.017,E2 -18144.017} C_VEL
LIN {X 0,Y 263.129,Z 362.708,A -85,B 0,C 180,E1 -18147.711,E2 -18147.711} C_VEL
LIN {X 0,Y 263.196,Z 362.698,A -85,B 0,C 180,E1 -18151.783,E2 -18151.783} C_VEL
LIN {X 0,Y 263.196,Z 362.701,A -85,B 0,C 180,E1 -18155.212,E2 -18155.212} C_VEL
LIN {X 0,Y 263.232,Z 362.694,A -85,B 0,C 180,E1 -18159.691,E2 -18159.691} C_VEL
LIN {X 0,Y 263.304,Z 362.685,A -85,B 0,C 180,E1 -18164.519,E2 -18164.519} C_VEL
LIN {X 0,Y 263.339,Z 362.681,A -85,B 0,C 180,E1 -18169.233,E2 -18169.233} C_VEL
LIN {X 0,Y 263.534,Z 362.656,A -85,B 0,C 180,E1 -18172.337,E2 -18172.337} C_VEL
LIN {X 0,Y 263.743,Z 362.63,A -85,B 0,C 180,E1 -18178.473,E2 -18178.473} C_VEL
LIN {X 0,Y 263.743,Z 362.63,A -85,B 0,C 180,E1 -18181.527,E2 -18181.527} C_VEL
LIN {X 0,Y 263.563,Z 362.652,A -85,B 0,C 180,E1 -18187.662,E2 -18187.662} C_VEL
LIN {X 0,Y 263.368,Z 362.68,A -85,B 0,C 180,E1 -18190.766,E2 -18190.766} C_VEL
LIN {X 0,Y 263.339,Z 362.68,A -85,B 0,C 180,E1 -18195.479,E2 -18195.479} C_VEL
LIN {X 0,Y 263.258,Z 362.693,A -85,B 0,C 180,E1 -18200.307,E2 -18200.307} C_VEL
LIN {X 0,Y 263.204,Z 362.697,A -85,B 0,C 180,E1 -18205.292,E2 -18205.292} C_VEL
LIN {X 0,Y 263.175,Z 362.701,A -85,B 0,C 180,E1 -18208.73,E2 -18208.73} C_VEL
LIN {X 0,Y 263.129,Z 362.709,A -85,B 0,C 180,E1 -18212.289,E2 -18212.289} C_VEL
LIN {X 0,Y 263.184,Z 362.701,A -85,B 0,C 180,E1 -18215.979,E2 -18215.979} C_VEL
LIN {X 0,Y 263.151,Z 362.704,A -85,B 0,C 180,E1 -18219.864,E2 -18219.864} C_VEL
LIN {X 0,Y 263.125,Z 362.71,A -85,B 0,C 180,E1 -18223.984,E2 -18223.984} C_VEL
LIN {X 0,Y 263.122,Z 362.709,A -85,B 0,C 180,E1 -18228.407,E2 -18228.407} C_VEL
LIN {X 0,Y 263.192,Z 362.698,A -85,B 0,C 180,E1 -18233.234,E2 -18233.234} C_VEL
LIN {X 0,Y 263.166,Z 362.703,A -85,B 0,C 180,E1 -18235.889,E2 -18235.889} C_VEL
LIN {X 0,Y 263.152,Z 362.705,A -85,B 0,C 180,E1 -18239.508,E2 -18239.508} C_VEL
LIN {X 0,Y 263.195,Z 362.696,A -85,B 0,C 180,E1 -18243.004,E2 -18243.004} C_VEL
LIN {X 0,Y 263.184,Z 362.7,A -85,B 0,C 180,E1 -18246.388,E2 -18246.388} C_VEL
LIN {X 0,Y 263.264,Z 362.693,A -85,B 0,C 180,E1 -18249.694,E2 -18249.694} C_VEL
LIN {X 0,Y 263.352,Z 362.678,A -85,B 0,C 180,E1 -18254.522,E2 -18254.522} C_VEL
LIN {X 0,Y 263.376,Z 362.675,A -85,B 0,C 180,E1 -18259.235,E2 -18259.235} C_VEL
LIN {X 0,Y 263.575,Z 362.651,A -85,B 0,C 180,E1 -18262.339,E2 -18262.339} C_VEL
LIN {X 0,Y 263.757,Z 362.628,A -85,B 0,C 180,E1 -18268.473,E2 -18268.473} C_VEL
LIN {X 0,Y 263.754,Z 362.632,A -85,B 0,C 180,E1 -18271.527,E2 -18271.527} C_VEL
LIN {X 0,Y 263.567,Z 362.655,A -85,B 0,C 180,E1 -18277.662,E2 -18277.662} C_VEL
LIN {X 0,Y 263.376,Z 362.676,A -85,B 0,C 180,E1 -18280.765,E2 -18280.765} C_VEL
LIN {X 0,Y 263.352,Z 362.681,A -85,B 0,C 180,E1 -18285.478,E2 -18285.478} C_VEL
LIN {X 0,Y 263.264,Z 362.689,A -85,B 0,C 180,E1 -18290.306,E2 -18290.306} C_VEL
LIN {X 0,Y 263.208,Z 362.7,A -85,B 0,C 180,E1 -18295.291,E2 -18295.291} C_VEL
LIN {X 0,Y 263.165,Z 362.703,A -85,B 0,C 180,E1 -18298.73,E2 -18298.73} C_VEL
LIN {X 0,Y 263.132,Z 362.707,A -85,B 0,C 180,E1 -18302.287,E2 -18302.287} C_VEL
LIN {X 0,Y 263.189,Z 362.7,A -85,B 0,C 180,E1 -18305.977,E2 -18305.977} C_VEL
LIN {X 0,Y 263.225,Z 362.885,A -85,B 0,C 180,E1 -18308.892,E2 -18308.892} C_VEL
LIN {X 0,Y 263.509,Z 364.093,A -85,B 0,C 180,E1 -18309.166,E2 -18309.166} C_VEL
LIN {X 0,Y 267.06,Z 375.974,A -85,B 0,C 180,E1 -18310.591,E2 -18310.591} C_VEL
LIN {X 0,Y 269.874,Z 386.648,A -85,B 0,C 180,E1 -18312.11,E2 -18312.11} C_VEL
LIN {X 0,Y 270.135,Z 387.948,A -85,B 0,C 180,E1 -18312.312,E2 -18312.312} C_VEL
LIN {X 0,Y 268.964,Z 399.536,A -85,B 0,C 180,E1 -18314.063,E2 -18314.063} C_VEL
LIN {X 0,Y 267.534,Z 410.522,A -85,B 0,C 180,E1 -18316.143,E2 -18316.143} C_VEL
LIN {X 0,Y 266.366,Z 419.64,A -85,B 0,C 180,E1 -18318.285,E2 -18318.285} C_VEL
LIN {X 0,Y 265.42,Z 427.38,A -85,B 0,C 180,E1 -18320.543,E2 -18320.543} C_VEL
LIN {X 0,Y 264.585,Z 433.749,A -85,B 0,C 180,E1 -18322.83,E2 -18322.83} C_VEL
LIN {X 0,Y 264.113,Z 438.571,A -85,B 0,C 180,E1 -18324.985,E2 -18324.985} C_VEL
LIN {X 0,Y 263.67,Z 443.417,A -85,B 0,C 180,E1 -18327.785,E2 -18327.785} C_VEL
LIN {X 0,Y 263.554,Z 445.658,A -85,B 0,C 180,E1 -18329.558,E2 -18329.558} C_VEL
LIN {X 0,Y 263.593,Z 447.6,A -85,B 0,C 180,E1 -18331.622,E2 -18331.622} C_VEL
LIN {X 0,Y 263.741,Z 448.508,A -85,B 0,C 180,E1 -18333.063,E2 -18333.063} C_VEL
LIN {X 0,Y 264.083,Z 449.159,A -85,B 0,C 180,E1 -18334.798,E2 -18334.798} C_VEL
LIN {X 0,Y 264.566,Z 449.252,A -85,B 0,C 180,E1 -18336.518,E2 -18336.518} C_VEL
LIN {X 0,Y 265.161,Z 448.882,A -85,B 0,C 180,E1 -18338.219,E2 -18338.219} C_VEL
LIN {X 0,Y 265.899,Z 448.024,A -85,B 0,C 180,E1 -18339.903,E2 -18339.903} C_VEL
LIN {X 0,Y 266.772,Z 446.663,A -85,B 0,C 180,E1 -18341.571,E2 -18341.571} C_VEL
LIN {X 0,Y 268.296,Z 443.728,A -85,B 0,C 180,E1 -18344.035,E2 -18344.035} C_VEL
LIN {X 0,Y 270.211,Z 439.583,A -85,B 0,C 180,E1 -18346.462,E2 -18346.462} C_VEL
LIN {X 0,Y 272.614,Z 433.705,A -85,B 0,C 180,E1 -18348.987,E2 -18348.987} C_VEL
LIN {X 0,Y 275.006,Z 427.175,A -85,B 0,C 180,E1 -18351.18,E2 -18351.18} C_VEL
LIN {X 0,Y 277.352,Z 420.087,A -85,B 0,C 180,E1 -18353.087,E2 -18353.087} C_VEL
LIN {X 0,Y 279.943,Z 411.445,A -85,B 0,C 180,E1 -18354.959,E2 -18354.959} C_VEL
LIN {X 0,Y 281.391,Z 405.479,A -85,B 0,C 180,E1 -18356.062,E2 -18356.062} C_VEL
LIN {X 0,Y 280.081,Z 398.418,A -85,B 0,C 180,E1 -18357.76,E2 -18357.76} C_VEL
LIN {X 0,Y 277.146,Z 389.072,A -85,B 0,C 180,E1 -18360,E2 -18360} C_VEL
LIN {X 0,Y 274.22,Z 381.533,A -85,B 0,C 180,E1 -18361.798,E2 -18361.798} C_VEL
LIN {X 0,Y 271.074,Z 375.526,A -85,B 0,C 180,E1 -18363.344,E2 -18363.344} C_VEL
LIN {X 0,Y 266.889,Z 368.888,A -85,B 0,C 180,E1 -18365.213,E2 -18365.213} C_VEL
LIN {X 0,Y 266.477,Z 367.94,A -85,B 0,C 180,E1 -18365.429,E2 -18365.429} C_VEL
LIN {X 0,Y 264.814,Z 365.97,A -85,B 0,C 180,E1 -18366.094,E2 -18366.094} C_VEL
LIN {X 0,Y 263.602,Z 363.335,A -85,B 0,C 180,E1 -18366.795,E2 -18366.795} C_VEL
LIN {X 0,Y 263.519,Z 362.696,A -85,B 0,C 180,E1 -18367.278,E2 -18367.278} C_VEL
LIN {X 0,Y 263.339,Z 362.683,A -85,B 0,C 180,E1 -18370.767,E2 -18370.767} C_VEL
LIN {X 0,Y 263.304,Z 362.686,A -85,B 0,C 180,E1 -18375.481,E2 -18375.481} C_VEL
LIN {X 0,Y 263.232,Z 362.688,A -85,B 0,C 180,E1 -18380.309,E2 -18380.309} C_VEL
LIN {X 0,Y 263.134,Z 362.706,A -85,B 0,C 180,E1 -18382.02,E2 -18382.02} C_VEL
LIN {X 0,Y 262.486,Z 363.011,A -85,B 0,C 180,E1 -18383.296,E2 -18383.296} C_VEL
LIN {X 0,Y 259.918,Z 364.468,A -85,B 0,C 180,E1 -18385.372,E2 -18385.372} C_VEL
LIN {X 0,Y 257.824,Z 365.994,A -85,B 0,C 180,E1 -18387.051,E2 -18387.051} C_VEL
LIN {X 0,Y 257.015,Z 367.06,A -85,B 0,C 180,E1 -18388.348,E2 -18388.348} C_VEL
LIN {X 0,Y 256.994,Z 367.362,A -85,B 0,C 180,E1 -18388.787,E2 -18388.787} C_VEL
LIN {X 0,Y 257.627,Z 370.551,A -85,B 0,C 180,E1 -18393.066,E2 -18393.066} C_VEL
LIN {X 0,Y 258.363,Z 373.916,A -85,B 0,C 180,E1 -18396.759,E2 -18396.759} C_VEL
LIN {X 0,Y 259.26,Z 378.099,A -85,B 0,C 180,E1 -18400.624,E2 -18400.624} C_VEL
LIN {X 0,Y 260.287,Z 383.096,A -85,B 0,C 180,E1 -18404.59,E2 -18404.59} C_VEL
LIN {X 0,Y 261.361,Z 389.265,A -85,B 0,C 180,E1 -18408.844,E2 -18408.844} C_VEL
LIN {X 0,Y 261.622,Z 392.176,A -85,B 0,C 180,E1 -18410.653,E2 -18410.653} C_VEL
LIN {X 0,Y 260.257,Z 397.9,A -85,B 0,C 180,E1 -18413.662,E2 -18413.662} C_VEL
LIN {X 0,Y 260.438,Z 399.974,A -85,B 0,C 180,E1 -18414.053,E2 -18414.053} C_VEL
LIN {X 0,Y 261.917,Z 404.948,A -85,B 0,C 180,E1 -18414.822,E2 -18414.822} C_VEL
LIN {X 0,Y 263.385,Z 411.082,A -85,B 0,C 180,E1 -18415.734,E2 -18415.734} C_VEL
LIN {X 0,Y 265.947,Z 423.91,A -85,B 0,C 180,E1 -18417.604,E2 -18417.604} C_VEL
LIN {X 0,Y 267.366,Z 437.534,A -85,B 0,C 180,E1 -18419.574,E2 -18419.574} C_VEL
LIN {X 0,Y 267.605,Z 448.029,A -85,B 0,C 180,E1 -18421.136,E2 -18421.136} C_VEL
LIN {X 0,Y 267.121,Z 458.366,A -85,B 0,C 180,E1 -18422.798,E2 -18422.798} C_VEL
LIN {X 0,Y 265.582,Z 469.435,A -85,B 0,C 180,E1 -18424.72,E2 -18424.72} C_VEL
LIN {X 0,Y 263.448,Z 479.853,A -85,B 0,C 180,E1 -18426.829,E2 -18426.829} C_VEL
LIN {X 0,Y 261.515,Z 487.755,A -85,B 0,C 180,E1 -18428.728,E2 -18428.728} C_VEL
LIN {X 0,Y 259.058,Z 495.772,A -85,B 0,C 180,E1 -18431.002,E2 -18431.002} C_VEL
LIN {X 0,Y 257.002,Z 503.298,A -85,B 0,C 180,E1 -18433.669,E2 -18433.669} C_VEL
LIN {X 0,Y 255.614,Z 509.526,A -85,B 0,C 180,E1 -18436.485,E2 -18436.485} C_VEL
LIN {X 0,Y 254.79,Z 514.738,A -85,B 0,C 180,E1 -18439.672,E2 -18439.672} C_VEL
LIN {X 0,Y 254.932,Z 518.415,A -85,B 0,C 180,E1 -18442.958,E2 -18442.958} C_VEL
LIN {X 0,Y 255.314,Z 519.964,A -85,B 0,C 180,E1 -18445.263,E2 -18445.263} C_VEL
LIN {X 0,Y 256.126,Z 520.663,A -85,B 0,C 180,E1 -18448.428,E2 -18448.428} C_VEL
LIN {X 0,Y 256.514,Z 520.373,A -85,B 0,C 180,E1 -18450,E2 -18450} C_VEL
LIN {X 0,Y 256.206,Z 519.545,A -85,B 0,C 180,E1 -18451.572,E2 -18451.572} C_VEL
LIN {X 0,Y 255.872,Z 518.221,A -85,B 0,C 180,E1 -18453.149,E2 -18453.149} C_VEL
LIN {X 0,Y 255.642,Z 515.395,A -85,B 0,C 180,E1 -18455.521,E2 -18455.521} C_VEL
LIN {X 0,Y 255.299,Z 511.372,A -85,B 0,C 180,E1 -18457.911,E2 -18457.911} C_VEL
LIN {X 0,Y 255.297,Z 505.128,A -85,B 0,C 180,E1 -18460.709,E2 -18460.709} C_VEL
LIN {X 0,Y 255.759,Z 498.283,A -85,B 0,C 180,E1 -18463.103,E2 -18463.103} C_VEL
LIN {X 0,Y 256.651,Z 489.692,A -85,B 0,C 180,E1 -18465.485,E2 -18465.485} C_VEL
LIN {X 0,Y 257.804,Z 480.968,A -85,B 0,C 180,E1 -18467.449,E2 -18467.449} C_VEL
LIN {X 0,Y 258.516,Z 474.792,A -85,B 0,C 180,E1 -18468.628,E2 -18468.628} C_VEL
LIN {X 0,Y 258.505,Z 463.285,A -85,B 0,C 180,E1 -18470.489,E2 -18470.489} C_VEL
LIN {X 0,Y 258.132,Z 451.345,A -85,B 0,C 180,E1 -18472.058,E2 -18472.058} C_VEL
LIN {X 0,Y 257.564,Z 438.235,A -85,B 0,C 180,E1 -18473.412,E2 -18473.412} C_VEL
LIN {X 0,Y 256.711,Z 424.68,A -85,B 0,C 180,E1 -18474.485,E2 -18474.485} C_VEL
LIN {X 0,Y 255.877,Z 414.078,A -85,B 0,C 180,E1 -18475.16,E2 -18475.16} C_VEL
LIN {X 0,Y 255.94,Z 413.135,A -85,B 0,C 180,E1 -18475.429,E2 -18475.429} C_VEL
LIN {X 0,Y 256.99,Z 404.585,A -85,B 0,C 180,E1 -18479.488,E2 -18479.488} C_VEL
LIN {X 0,Y 258.462,Z 395.412,A -85,B 0,C 180,E1 -18483.877,E2 -18483.877} C_VEL
LIN {X 0,Y 259.927,Z 387.942,A -85,B 0,C 180,E1 -18487.47,E2 -18487.47} C_VEL
LIN {X 0,Y 260.239,Z 385.957,A -85,B 0,C 180,E1 -18488.448,E2 -18488.448} C_VEL
LIN {X 0,Y 259.61,Z 381.561,A -85,B 0,C 180,E1 -18490.712,E2 -18490.712} C_VEL
LIN {X 0,Y 258.004,Z 373.429,A -85,B 0,C 180,E1 -18495.09,E2 -18495.09} C_VEL
LIN {X 0,Y 256.455,Z 365.447,A -85,B 0,C 180,E1 -18499.631,E2 -18499.631} C_VEL
LIN {X 0,Y 256.102,Z 363.622,A -85,B 0,C 180,E1 -18500.863,E2 -18500.863} C_VEL
LIN {X 0,Y 256.076,Z 363.587,A -85,B 0,C 180,E1 -18504.806,E2 -18504.806} C_VEL
LIN {X 0,Y 256.088,Z 363.584,A -85,B 0,C 180,E1 -18508.572,E2 -18508.572} C_VEL
LIN {X 0,Y 256.137,Z 363.577,A -85,B 0,C 180,E1 -18512.195,E2 -18512.195} C_VEL
LIN {X 0,Y 256.137,Z 363.577,A -85,B 0,C 180,E1 -18515.696,E2 -18515.696} C_VEL
LIN {X 0,Y 256.143,Z 363.579,A -85,B 0,C 180,E1 -18519.103,E2 -18519.103} C_VEL
LIN {X 0,Y 256.239,Z 363.564,A -85,B 0,C 180,E1 -18524.081,E2 -18524.081} C_VEL
LIN {X 0,Y 256.281,Z 363.56,A -85,B 0,C 180,E1 -18528.933,E2 -18528.933} C_VEL
LIN {X 0,Y 256.495,Z 363.533,A -85,B 0,C 180,E1 -18532.126,E2 -18532.126} C_VEL
LIN {X 0,Y 256.487,Z 363.536,A -85,B 0,C 180,E1 -18536.858,E2 -18536.858} C_VEL
LIN {X 0,Y 256.758,Z 363.5,A -85,B 0,C 180,E1 -18540,E2 -18540} C_VEL
LIN {X 0,Y 256.488,Z 363.534,A -85,B 0,C 180,E1 -18543.141,E2 -18543.141} C_VEL
LIN {X 0,Y 256.531,Z 363.528,A -85,B 0,C 180,E1 -18547.873,E2 -18547.873} C_VEL
LIN {X 0,Y 256.303,Z 363.557,A -85,B 0,C 180,E1 -18551.066,E2 -18551.066} C_VEL
LIN {X 0,Y 256.289,Z 363.558,A -85,B 0,C 180,E1 -18555.916,E2 -18555.916} C_VEL
LIN {X 0,Y 256.161,Z 363.574,A -85,B 0,C 180,E1 -18560.896,E2 -18560.896} C_VEL
LIN {X 0,Y 256.184,Z 363.572,A -85,B 0,C 180,E1 -18565.139,E2 -18565.139} C_VEL
LIN {X 0,Y 256.11,Z 363.579,A -85,B 0,C 180,E1 -18569.6,E2 -18569.6} C_VEL
LIN {X 0,Y 256.081,Z 363.584,A -85,B 0,C 180,E1 -18573.291,E2 -18573.291} C_VEL
LIN {X 0,Y 256.135,Z 363.576,A -85,B 0,C 180,E1 -18577.279,E2 -18577.279} C_VEL
LIN {X 0,Y 256.079,Z 363.584,A -85,B 0,C 180,E1 -18581.199,E2 -18581.199} C_VEL
LIN {X 0,Y 256.057,Z 363.587,A -85,B 0,C 180,E1 -18585.531,E2 -18585.531} C_VEL
LIN {X 0,Y 256.052,Z 363.588,A -85,B 0,C 180,E1 -18588.797,E2 -18588.797} C_VEL
LIN {X 0,Y 256.137,Z 363.576,A -85,B 0,C 180,E1 -18592.87,E2 -18592.87} C_VEL
LIN {X 0,Y 256.076,Z 363.585,A -85,B 0,C 180,E1 -18596.709,E2 -18596.709} C_VEL
LIN {X 0,Y 256.142,Z 363.577,A -85,B 0,C 180,E1 -18601.404,E2 -18601.404} C_VEL
LIN {X 0,Y 256.168,Z 363.576,A -85,B 0,C 180,E1 -18605.7,E2 -18605.7} C_VEL
LIN {X 0,Y 256.167,Z 363.573,A -85,B 0,C 180,E1 -18609.106,E2 -18609.106} C_VEL
LIN {X 0,Y 256.301,Z 363.559,A -85,B 0,C 180,E1 -18614.086,E2 -18614.086} C_VEL
LIN {X 0,Y 256.311,Z 363.554,A -85,B 0,C 180,E1 -18618.934,E2 -18618.934} C_VEL
LIN {X 0,Y 256.542,Z 363.528,A -85,B 0,C 180,E1 -18622.127,E2 -18622.127} C_VEL
LIN {X 0,Y 256.719,Z 363.504,A -85,B 0,C 180,E1 -18628.431,E2 -18628.431} C_VEL
LIN {X 0,Y 256.717,Z 363.508,A -85,B 0,C 180,E1 -18631.569,E2 -18631.569} C_VEL
LIN {X 0,Y 256.485,Z 363.532,A -85,B 0,C 180,E1 -18636.292,E2 -18636.292} C_VEL
LIN {X 0,Y 256.452,Z 363.542,A -85,B 0,C 180,E1 -18639.464,E2 -18639.464} C_VEL
LIN {X 0,Y 256.257,Z 363.562,A -85,B 0,C 180,E1 -18644.29,E2 -18644.29} C_VEL
LIN {X 0,Y 256.212,Z 363.571,A -85,B 0,C 180,E1 -18647.561,E2 -18647.561} C_VEL
LIN {X 0,Y 256.158,Z 363.578,A -85,B 0,C 180,E1 -18651.119,E2 -18651.119} C_VEL
LIN {X 0,Y 256.188,Z 363.575,A -85,B 0,C 180,E1 -18655.138,E2 -18655.138} C_VEL
LIN {X 0,Y 256.103,Z 363.584,A -85,B 0,C 180,E1 -18659.6,E2 -18659.6} C_VEL
LIN {X 0,Y 256.084,Z 363.587,A -85,B 0,C 180,E1 -18663.289,E2 -18663.289} C_VEL
LIN {X 0,Y 256.144,Z 363.58,A -85,B 0,C 180,E1 -18667.279,E2 -18667.279} C_VEL
LIN {X 0,Y 256.175,Z 363.711,A -85,B 0,C 180,E1 -18668.436,E2 -18668.436} C_VEL
LIN {X 0,Y 256.425,Z 364.818,A -85,B 0,C 180,E1 -18668.733,E2 -18668.733} C_VEL
LIN {X 0,Y 260.318,Z 378.022,A -85,B 0,C 180,E1 -18670.386,E2 -18670.386} C_VEL
LIN {X 0,Y 263.017,Z 388.343,A -85,B 0,C 180,E1 -18671.913,E2 -18671.913} C_VEL
LIN {X 0,Y 263.06,Z 391.337,A -85,B 0,C 180,E1 -18672.353,E2 -18672.353} C_VEL
LIN {X 0,Y 261.854,Z 401.698,A -85,B 0,C 180,E1 -18674.023,E2 -18674.023} C_VEL
LIN {X 0,Y 260.565,Z 411.229,A -85,B 0,C 180,E1 -18675.889,E2 -18675.889} C_VEL
LIN {X 0,Y 259.463,Z 419.693,A -85,B 0,C 180,E1 -18677.902,E2 -18677.902} C_VEL
LIN {X 0,Y 258.394,Z 428.121,A -85,B 0,C 180,E1 -18680.376,E2 -18680.376} C_VEL
LIN {X 0,Y 257.431,Z 435.442,A -85,B 0,C 180,E1 -18683.086,E2 -18683.086} C_VEL
LIN {X 0,Y 256.825,Z 441.358,A -85,B 0,C 180,E1 -18685.962,E2 -18685.962} C_VEL
LIN {X 0,Y 256.586,Z 445.433,A -85,B 0,C 180,E1 -18688.64,E2 -18688.64} C_VEL
LIN {X 0,Y 256.539,Z 448.199,A -85,B 0,C 180,E1 -18691.239,E2 -18691.239} C_VEL
LIN {X 0,Y 256.984,Z 450.061,A -85,B 0,C 180,E1 -18694.483,E2 -18694.483} C_VEL
LIN {X 0,Y 257.905,Z 450.294,A -85,B 0,C 180,E1 -18697.573,E2 -18697.573} C_VEL
LIN {X 0,Y 258.613,Z 449.72,A -85,B 0,C 180,E1 -18699.312,E2 -18699.312} C_VEL
LIN {X 0,Y 259.648,Z 448.47,A -85,B 0,C 180,E1 -18701.323,E2 -18701.323} C_VEL
LIN {X 0,Y 260.985,Z 446.215,A -85,B 0,C 180,E1 -18703.575,E2 -18703.575} C_VEL
LIN {X 0,Y 262.888,Z 442.584,A -85,B 0,C 180,E1 -18706.078,E2 -18706.078} C_VEL
LIN {X 0,Y 265.256,Z 437.501,A -85,B 0,C 180,E1 -18708.607,E2 -18708.607} C_VEL
LIN {X 0,Y 267.697,Z 431.433,A -85,B 0,C 180,E1 -18710.937,E2 -18710.937} C_VEL
LIN {X 0,Y 270.102,Z 424.966,A -85,B 0,C 180,E1 -18712.9,E2 -18712.9} C_VEL
LIN {X 0,Y 272.717,Z 417.17,A -85,B 0,C 180,E1 -18714.825,E2 -18714.825} C_VEL
LIN {X 0,Y 275.384,Z 408.165,A -85,B 0,C 180,E1 -18716.626,E2 -18716.626} C_VEL
LIN {X 0,Y 274.635,Z 403.287,A -85,B 0,C 180,E1 -18717.874,E2 -18717.874} C_VEL
LIN {X 0,Y 271.521,Z 392.104,A -85,B 0,C 180,E1 -18720.738,E2 -18720.738} C_VEL
LIN {X 0,Y 268.815,Z 384.932,A -85,B 0,C 180,E1 -18722.572,E2 -18722.572} C_VEL
LIN {X 0,Y 265.142,Z 377.981,A -85,B 0,C 180,E1 -18724.561,E2 -18724.561} C_VEL
LIN {X 0,Y 260.3,Z 370.145,A -85,B 0,C 180,E1 -18726.978,E2 -18726.978} C_VEL
LIN {X 0,Y 259.188,Z 368.258,A -85,B 0,C 180,E1 -18727.547,E2 -18727.547} C_VEL
LIN {X 0,Y 257.291,Z 366.106,A -85,B 0,C 180,E1 -18728.393,E2 -18728.393} C_VEL
LIN {X 0,Y 256.549,Z 364.181,A -85,B 0,C 180,E1 -18728.963,E2 -18728.963} C_VEL
LIN {X 0,Y 256.397,Z 363.563,A -85,B 0,C 180,E1 -18729.665,E2 -18729.665} C_VEL
LIN {X 0,Y 256.225,Z 363.569,A -85,B 0,C 180,E1 -18734.292,E2 -18734.292} C_VEL
LIN {X 0,Y 256.167,Z 363.566,A -85,B 0,C 180,E1 -18737.565,E2 -18737.565} C_VEL
LIN {X 0,Y 256.132,Z 363.641,A -85,B 0,C 180,E1 -18741.339,E2 -18741.339} C_VEL
LIN {X 0,Y 256.626,Z 365.712,A -85,B 0,C 180,E1 -18745.988,E2 -18745.988} C_VEL
LIN {X 0,Y 256.994,Z 367.362,A -85,B 0,C 180,E1 -18748.787,E2 -18748.787} C_VEL
LIN {X 0,Y 256.527,Z 368.462,A -85,B 0,C 180,E1 -18750.076,E2 -18750.076} C_VEL
LIN {X 0,Y 254.095,Z 370.969,A -85,B 0,C 180,E1 -18752.159,E2 -18752.159} C_VEL
LIN {X 0,Y 252.065,Z 373.144,A -85,B 0,C 180,E1 -18753.845,E2 -18753.845} C_VEL
LIN {X 0,Y 251.342,Z 374.611,A -85,B 0,C 180,E1 -18755.153,E2 -18755.153} C_VEL
LIN {X 0,Y 251.365,Z 375.032,A -85,B 0,C 180,E1 -18755.596,E2 -18755.596} C_VEL
LIN {X 0,Y 252.324,Z 379.318,A -85,B 0,C 180,E1 -18759.838,E2 -18759.838} C_VEL
LIN {X 0,Y 253.295,Z 384.2,A -85,B 0,C 180,E1 -18763.921,E2 -18763.921} C_VEL
LIN {X 0,Y 254.092,Z 388.576,A -85,B 0,C 180,E1 -18767.135,E2 -18767.135} C_VEL
LIN {X 0,Y 254.642,Z 392.197,A -85,B 0,C 180,E1 -18769.567,E2 -18769.567} C_VEL
LIN {X 0,Y 254.691,Z 393.865,A -85,B 0,C 180,E1 -18770.606,E2 -18770.606} C_VEL
LIN {X 0,Y 254.146,Z 396.335,A -85,B 0,C 180,E1 -18771.839,E2 -18771.839} C_VEL
LIN {X 0,Y 254.976,Z 400.533,A -85,B 0,C 180,E1 -18772.582,E2 -18772.582} C_VEL
LIN {X 0,Y 255.901,Z 403.261,A -85,B 0,C 180,E1 -18773.092,E2 -18773.092} C_VEL
LIN {X 0,Y 258.285,Z 413.219,A -85,B 0,C 180,E1 -18774.717,E2 -18774.717} C_VEL
LIN {X 0,Y 260.453,Z 426.377,A -85,B 0,C 180,E1 -18776.772,E2 -18776.772} C_VEL
LIN {X 0,Y 261.497,Z 438.348,A -85,B 0,C 180,E1 -18778.627,E2 -18778.627} C_VEL
LIN {X 0,Y 261.469,Z 450.543,A -85,B 0,C 180,E1 -18780.575,E2 -18780.575} C_VEL
LIN {X 0,Y 260.728,Z 460.548,A -85,B 0,C 180,E1 -18782.292,E2 -18782.292} C_VEL
LIN {X 0,Y 258.961,Z 470.994,A -85,B 0,C 180,E1 -18784.265,E2 -18784.265} C_VEL
LIN {X 0,Y 256.509,Z 481.646,A -85,B 0,C 180,E1 -18786.592,E2 -18786.592} C_VEL
LIN {X 0,Y 254.445,Z 489.109,A -85,B 0,C 180,E1 -18788.533,E2 -18788.533} C_VEL
LIN {X 0,Y 251.967,Z 496.682,A -85,B 0,C 180,E1 -18790.869,E2 -18790.869} C_VEL
LIN {X 0,Y 250.15,Z 502.267,A -85,B 0,C 180,E1 -18792.97,E2 -18792.97} C_VEL
LIN {X 0,Y 248.969,Z 507.324,A -85,B 0,C 180,E1 -18795.283,E2 -18795.283} C_VEL
LIN {X 0,Y 248.058,Z 511.617,A -85,B 0,C 180,E1 -18797.732,E2 -18797.732} C_VEL
LIN {X 0,Y 247.699,Z 514.96,A -85,B 0,C 180,E1 -18800.199,E2 -18800.199} C_VEL
LIN {X 0,Y 247.943,Z 518.034,A -85,B 0,C 180,E1 -18803.49,E2 -18803.49} C_VEL
LIN {X 0,Y 248.24,Z 518.95,A -85,B 0,C 180,E1 -18805.128,E2 -18805.128} C_VEL
LIN {X 0,Y 249.082,Z 519.538,A -85,B 0,C 180,E1 -18808.383,E2 -18808.383} C_VEL
LIN {X 0,Y 249.49,Z 519.214,A -85,B 0,C 180,E1 -18810,E2 -18810} C_VEL
LIN {X 0,Y 249.173,Z 518.315,A -85,B 0,C 180,E1 -18811.616,E2 -18811.616} C_VEL
LIN {X 0,Y 248.841,Z 516.925,A -85,B 0,C 180,E1 -18813.238,E2 -18813.238} C_VEL
LIN {X 0,Y 248.602,Z 514.004,A -85,B 0,C 180,E1 -18815.678,E2 -18815.678} C_VEL
LIN {X 0,Y 248.24,Z 509.875,A -85,B 0,C 180,E1 -18818.138,E2 -18818.138} C_VEL
LIN {X 0,Y 248.292,Z 503.517,A -85,B 0,C 180,E1 -18821.014,E2 -18821.014} C_VEL
LIN {X 0,Y 248.83,Z 496.487,A -85,B 0,C 180,E1 -18823.474,E2 -18823.474} C_VEL
LIN {X 0,Y 249.766,Z 487.738,A -85,B 0,C 180,E1 -18825.923,E2 -18825.923} C_VEL
LIN {X 0,Y 251.163,Z 477.821,A -85,B 0,C 180,E1 -18828.137,E2 -18828.137} C_VEL
LIN {X 0,Y 251.441,Z 472.346,A -85,B 0,C 180,E1 -18829.173,E2 -18829.173} C_VEL
LIN {X 0,Y 251.362,Z 461.93,A -85,B 0,C 180,E1 -18830.884,E2 -18830.884} C_VEL
LIN {X 0,Y 251.048,Z 449.801,A -85,B 0,C 180,E1 -18832.508,E2 -18832.508} C_VEL
LIN {X 0,Y 250.503,Z 436.634,A -85,B 0,C 180,E1 -18833.894,E2 -18833.894} C_VEL
LIN {X 0,Y 249.639,Z 423.039,A -85,B 0,C 180,E1 -18834.979,E2 -18834.979} C_VEL
LIN {X 0,Y 248.893,Z 412.958,A -85,B 0,C 180,E1 -18835.638,E2 -18835.638} C_VEL
LIN {X 0,Y 249.958,Z 404.31,A -85,B 0,C 180,E1 -18839.775,E2 -18839.775} C_VEL
LIN {X 0,Y 251.41,Z 395.763,A -85,B 0,C 180,E1 -18843.992,E2 -18843.992} C_VEL
LIN {X 0,Y 253.103,Z 387.108,A -85,B 0,C 180,E1 -18848.315,E2 -18848.315} C_VEL
LIN {X 0,Y 252.958,Z 384.402,A -85,B 0,C 180,E1 -18849.717,E2 -18849.717} C_VEL
LIN {X 0,Y 251.595,Z 377.59,A -85,B 0,C 180,E1 -18853.424,E2 -18853.424} C_VEL
LIN {X 0,Y 250.156,Z 370.255,A -85,B 0,C 180,E1 -18857.602,E2 -18857.602} C_VEL
LIN {X 0,Y 249.047,Z 364.528,A -85,B 0,C 180,E1 -18861.105,E2 -18861.105} C_VEL
LIN {X 0,Y 249.039,Z 364.464,A -85,B 0,C 180,E1 -18865.639,E2 -18865.639} C_VEL
LIN {X 0,Y 249.048,Z 364.462,A -85,B 0,C 180,E1 -18869.472,E2 -18869.472} C_VEL
LIN {X 0,Y 249.065,Z 364.462,A -85,B 0,C 180,E1 -18873.161,E2 -18873.161} C_VEL
LIN {X 0,Y 249.055,Z 364.46,A -85,B 0,C 180,E1 -18876.73,E2 -18876.73} C_VEL
LIN {X 0,Y 249.077,Z 364.456,A -85,B 0,C 180,E1 -18880.209,E2 -18880.209} C_VEL
LIN {X 0,Y 249.191,Z 364.442,A -85,B 0,C 180,E1 -18883.618,E2 -18883.618} C_VEL
LIN {X 0,Y 249.224,Z 364.437,A -85,B 0,C 180,E1 -18888.615,E2 -18888.615} C_VEL
LIN {X 0,Y 249.434,Z 364.412,A -85,B 0,C 180,E1 -18891.901,E2 -18891.901} C_VEL
LIN {X 0,Y 249.281,Z 364.432,A -85,B 0,C 180,E1 -18895.148,E2 -18895.148} C_VEL
LIN {X 0,Y 249.668,Z 364.383,A -85,B 0,C 180,E1 -18898.387,E2 -18898.387} C_VEL
LIN {X 0,Y 249.668,Z 364.383,A -85,B 0,C 180,E1 -18901.613,E2 -18901.613} C_VEL
LIN {X 0,Y 249.439,Z 364.41,A -85,B 0,C 180,E1 -18906.824,E2 -18906.824} C_VEL
LIN {X 0,Y 249.384,Z 364.418,A -85,B 0,C 180,E1 -18909.735,E2 -18909.735} C_VEL
LIN {X 0,Y 249.195,Z 364.445,A -85,B 0,C 180,E1 -18914.704,E2 -18914.704} C_VEL
LIN {X 0,Y 249.134,Z 364.451,A -85,B 0,C 180,E1 -18918.078,E2 -18918.078} C_VEL
LIN {X 0,Y 249.082,Z 364.454,A -85,B 0,C 180,E1 -18921.519,E2 -18921.519} C_VEL
LIN {X 0,Y 249.126,Z 364.451,A -85,B 0,C 180,E1 -18925.483,E2 -18925.483} C_VEL
LIN {X 0,Y 249.079,Z 364.455,A -85,B 0,C 180,E1 -18928.994,E2 -18928.994} C_VEL
LIN {X 0,Y 249.032,Z 364.466,A -85,B 0,C 180,E1 -18932.426,E2 -18932.426} C_VEL
LIN {X 0,Y 249.07,Z 364.46,A -85,B 0,C 180,E1 -18936.339,E2 -18936.339} C_VEL
LIN {X 0,Y 249.041,Z 364.464,A -85,B 0,C 180,E1 -18940.471,E2 -18940.471} C_VEL
LIN {X 0,Y 249.003,Z 364.465,A -85,B 0,C 180,E1 -18944.879,E2 -18944.879} C_VEL
LIN {X 0,Y 249.014,Z 364.463,A -85,B 0,C 180,E1 -18947.364,E2 -18947.364} C_VEL
LIN {X 0,Y 249.047,Z 364.463,A -85,B 0,C 180,E1 -18952.2,E2 -18952.2} C_VEL
LIN {X 0,Y 249.057,Z 364.459,A -85,B 0,C 180,E1 -18955.643,E2 -18955.643} C_VEL
LIN {X 0,Y 249.053,Z 364.461,A -85,B 0,C 180,E1 -18959.474,E2 -18959.474} C_VEL
LIN {X 0,Y 249.076,Z 364.455,A -85,B 0,C 180,E1 -18963.163,E2 -18963.163} C_VEL
LIN {X 0,Y 249.08,Z 364.456,A -85,B 0,C 180,E1 -18966.733,E2 -18966.733} C_VEL
LIN {X 0,Y 249.112,Z 364.452,A -85,B 0,C 180,E1 -18970.212,E2 -18970.212} C_VEL
LIN {X 0,Y 249.243,Z 364.438,A -85,B 0,C 180,E1 -18973.622,E2 -18973.622} C_VEL
LIN {X 0,Y 249.255,Z 364.433,A -85,B 0,C 180,E1 -18978.617,E2 -18978.617} C_VEL
LIN {X 0,Y 249.486,Z 364.408,A -85,B 0,C 180,E1 -18981.903,E2 -18981.903} C_VEL
LIN {X 0,Y 249.443,Z 364.41,A -85,B 0,C 180,E1 -18986.77,E2 -18986.77} C_VEL
LIN {X 0,Y 249.738,Z 364.376,A -85,B 0,C 180,E1 -18990,E2 -18990} C_VEL
LIN {X 0,Y 249.439,Z 364.413,A -85,B 0,C 180,E1 -18993.23,E2 -18993.23} C_VEL
LIN {X 0,Y 249.471,Z 364.408,A -85,B 0,C 180,E1 -18998.097,E2 -18998.097} C_VEL
LIN {X 0,Y 249.255,Z 364.436,A -85,B 0,C 180,E1 -19001.383,E2 -19001.383} C_VEL
LIN {X 0,Y 249.243,Z 364.436,A -85,B 0,C 180,E1 -19006.378,E2 -19006.378} C_VEL
LIN {X 0,Y 249.088,Z 364.458,A -85,B 0,C 180,E1 -19011.517,E2 -19011.517} C_VEL
LIN {X 0,Y 249.13,Z 364.452,A -85,B 0,C 180,E1 -19015.481,E2 -19015.481} C_VEL
LIN {X 0,Y 249.073,Z 364.461,A -85,B 0,C 180,E1 -19018.988,E2 -19018.988} C_VEL
LIN {X 0,Y 249.035,Z 364.464,A -85,B 0,C 180,E1 -19022.424,E2 -19022.424} C_VEL
LIN {X 0,Y 249.074,Z 364.459,A -85,B 0,C 180,E1 -19026.337,E2 -19026.337} C_VEL
LIN {X 0,Y 249.138,Z 364.602,A -85,B 0,C 180,E1 -19028.016,E2 -19028.016} C_VEL
LIN {X 0,Y 249.385,Z 365.728,A -85,B 0,C 180,E1 -19028.314,E2 -19028.314} C_VEL
LIN {X 0,Y 253.064,Z 378.137,A -85,B 0,C 180,E1 -19029.9,E2 -19029.9} C_VEL
LIN {X 0,Y 255.944,Z 389.115,A -85,B 0,C 180,E1 -19031.562,E2 -19031.562} C_VEL
LIN {X 0,Y 256.22,Z 391.411,A -85,B 0,C 180,E1 -19031.925,E2 -19031.925} C_VEL
LIN {X 0,Y 255.068,Z 401.412,A -85,B 0,C 180,E1 -19033.537,E2 -19033.537} C_VEL
LIN {X 0,Y 253.634,Z 411.834,A -85,B 0,C 180,E1 -19035.6,E2 -19035.6} C_VEL
LIN {X 0,Y 252.528,Z 419.942,A -85,B 0,C 180,E1 -19037.554,E2 -19037.554} C_VEL
LIN {X 0,Y 251.464,Z 428.271,A -85,B 0,C 180,E1 -19039.998,E2 -19039.998} C_VEL
LIN {X 0,Y 250.552,Z 434.859,A -85,B 0,C 180,E1 -19042.404,E2 -19042.404} C_VEL
LIN {X 0,Y 249.927,Z 440.842,A -85,B 0,C 180,E1 -19045.177,E2 -19045.177} C_VEL
LIN {X 0,Y 249.597,Z 444.955,A -85,B 0,C 180,E1 -19047.657,E2 -19047.657} C_VEL
LIN {X 0,Y 249.496,Z 447.368,A -85,B 0,C 180,E1 -19049.533,E2 -19049.533} C_VEL
LIN {X 0,Y 249.521,Z 449.191,A -85,B 0,C 180,E1 -19051.391,E2 -19051.391} C_VEL
LIN {X 0,Y 249.901,Z 450.929,A -85,B 0,C 180,E1 -19054.147,E2 -19054.147} C_VEL
LIN {X 0,Y 250.896,Z 451.44,A -85,B 0,C 180,E1 -19057.572,E2 -19057.572} C_VEL
LIN {X 0,Y 252.173,Z 450.507,A -85,B 0,C 180,E1 -19060.462,E2 -19060.462} C_VEL
LIN {X 0,Y 253.158,Z 449.281,A -85,B 0,C 180,E1 -19062.219,E2 -19062.219} C_VEL
LIN {X 0,Y 254.871,Z 446.548,A -85,B 0,C 180,E1 -19064.817,E2 -19064.817} C_VEL
LIN {X 0,Y 256.999,Z 442.636,A -85,B 0,C 180,E1 -19067.363,E2 -19067.363} C_VEL
LIN {X 0,Y 259.558,Z 437.42,A -85,B 0,C 180,E1 -19069.863,E2 -19069.863} C_VEL
LIN {X 0,Y 262.381,Z 430.73,A -85,B 0,C 180,E1 -19072.324,E2 -19072.324} C_VEL
LIN {X 0,Y 265.529,Z 422.493,A -85,B 0,C 180,E1 -19074.685,E2 -19074.685} C_VEL
LIN {X 0,Y 268.623,Z 413.2,A -85,B 0,C 180,E1 -19076.771,E2 -19076.771} C_VEL
LIN {X 0,Y 269.34,Z 410.162,A -85,B 0,C 180,E1 -19077.407,E2 -19077.407} C_VEL
LIN {X 0,Y 268.101,Z 403.523,A -85,B 0,C 180,E1 -19079.249,E2 -19079.249} C_VEL
LIN {X 0,Y 265.489,Z 393.918,A -85,B 0,C 180,E1 -19081.845,E2 -19081.845} C_VEL
LIN {X 0,Y 263.003,Z 387.543,A -85,B 0,C 180,E1 -19083.665,E2 -19083.665} C_VEL
LIN {X 0,Y 257.92,Z 378.156,A -85,B 0,C 180,E1 -19086.65,E2 -19086.65} C_VEL
LIN {X 0,Y 255.498,Z 374.048,A -85,B 0,C 180,E1 -19088.016,E2 -19088.016} C_VEL
LIN {X 0,Y 253.592,Z 371.351,A -85,B 0,C 180,E1 -19089.068,E2 -19089.068} C_VEL
LIN {X 0,Y 252.439,Z 369.454,A -85,B 0,C 180,E1 -19089.727,E2 -19089.727} C_VEL
LIN {X 0,Y 250.19,Z 367.145,A -85,B 0,C 180,E1 -19090.889,E2 -19090.889} C_VEL
LIN {X 0,Y 249.327,Z 365.12,A -85,B 0,C 180,E1 -19091.586,E2 -19091.586} C_VEL
LIN {X 0,Y 249.204,Z 364.479,A -85,B 0,C 180,E1 -19092.211,E2 -19092.211} C_VEL
LIN {X 0,Y 249.19,Z 364.61,A -85,B 0,C 180,E1 -19096.486,E2 -19096.486} C_VEL
LIN {X 0,Y 249.425,Z 366.065,A -85,B 0,C 180,E1 -19101.595,E2 -19101.595} C_VEL
LIN {X 0,Y 250.021,Z 368.429,A -85,B 0,C 180,E1 -19106.728,E2 -19106.728} C_VEL
LIN {X 0,Y 250.456,Z 370.739,A -85,B 0,C 180,E1 -19110.338,E2 -19110.338} C_VEL
LIN {X 0,Y 251.09,Z 373.641,A -85,B 0,C 180,E1 -19114.042,E2 -19114.042} C_VEL
LIN {X 0,Y 251.365,Z 375.032,A -85,B 0,C 180,E1 -19115.596,E2 -19115.596} C_VEL
LIN {X 0,Y 251.034,Z 376.466,A -85,B 0,C 180,E1 -19116.898,E2 -19116.898} C_VEL
LIN {X 0,Y 248.77,Z 379.47,A -85,B 0,C 180,E1 -19118.999,E2 -19118.999} C_VEL
LIN {X 0,Y 246.814,Z 382.055,A -85,B 0,C 180,E1 -19120.696,E2 -19120.696} C_VEL
LIN {X 0,Y 246.11,Z 383.87,A -85,B 0,C 180,E1 -19122.01,E2 -19122.01} C_VEL
LIN {X 0,Y 246.133,Z 384.42,A -85,B 0,C 180,E1 -19122.456,E2 -19122.456} C_VEL
LIN {X 0,Y 247.015,Z 389.15,A -85,B 0,C 180,E1 -19126.179,E2 -19126.179} C_VEL
LIN {X 0,Y 247.801,Z 394.067,A -85,B 0,C 180,E1 -19129.488,E2 -19129.488} C_VEL
LIN {X 0,Y 248.313,Z 396.281,A -85,B 0,C 180,E1 -19130.03,E2 -19130.03} C_VEL
LIN {X 0,Y 249.998,Z 401.339,A -85,B 0,C 180,E1 -19131.113,E2 -19131.113} C_VEL
LIN {X 0,Y 251.113,Z 405.831,A -85,B 0,C 180,E1 -19131.943,E2 -19131.943} C_VEL
LIN {X 0,Y 253.376,Z 416.779,A -85,B 0,C 180,E1 -19133.887,E2 -19133.887} C_VEL
LIN {X 0,Y 255.059,Z 429.537,A -85,B 0,C 180,E1 -19136.022,E2 -19136.022} C_VEL
LIN {X 0,Y 255.717,Z 441.857,A -85,B 0,C 180,E1 -19138.078,E2 -19138.078} C_VEL
LIN {X 0,Y 255.306,Z 453.18,A -85,B 0,C 180,E1 -19140.027,E2 -19140.027} C_VEL
LIN {X 0,Y 254.172,Z 463.597,A -85,B 0,C 180,E1 -19141.963,E2 -19141.963} C_VEL
LIN {X 0,Y 252.15,Z 473.397,A -85,B 0,C 180,E1 -19143.961,E2 -19143.961} C_VEL
LIN {X 0,Y 249.556,Z 483.299,A -85,B 0,C 180,E1 -19146.341,E2 -19146.341} C_VEL
LIN {X 0,Y 246.85,Z 491.64,A -85,B 0,C 180,E1 -19148.716,E2 -19148.716} C_VEL
LIN {X 0,Y 244.161,Z 499.595,A -85,B 0,C 180,E1 -19151.541,E2 -19151.541} C_VEL
LIN {X 0,Y 242.96,Z 503.397,A -85,B 0,C 180,E1 -19153.186,E2 -19153.186} C_VEL
LIN {X 0,Y 241.678,Z 508.229,A -85,B 0,C 180,E1 -19155.69,E2 -19155.69} C_VEL
LIN {X 0,Y 240.869,Z 512.083,A -85,B 0,C 180,E1 -19158.215,E2 -19158.215} C_VEL
LIN {X 0,Y 240.632,Z 515.811,A -85,B 0,C 180,E1 -19161.603,E2 -19161.603} C_VEL
LIN {X 0,Y 240.858,Z 517.071,A -85,B 0,C 180,E1 -19163.298,E2 -19163.298} C_VEL
LIN {X 0,Y 241.168,Z 517.919,A -85,B 0,C 180,E1 -19164.985,E2 -19164.985} C_VEL
LIN {X 0,Y 242.036,Z 518.422,A -85,B 0,C 180,E1 -19168.336,E2 -19168.336} C_VEL
LIN {X 0,Y 242.466,Z 518.037,A -85,B 0,C 180,E1 -19170,E2 -19170} C_VEL
LIN {X 0,Y 242.141,Z 517.044,A -85,B 0,C 180,E1 -19171.663,E2 -19171.663} C_VEL
LIN {X 0,Y 241.812,Z 515.602,A -85,B 0,C 180,E1 -19173.332,E2 -19173.332} C_VEL
LIN {X 0,Y 241.555,Z 512.562,A -85,B 0,C 180,E1 -19175.845,E2 -19175.845} C_VEL
LIN {X 0,Y 241.185,Z 508.306,A -85,B 0,C 180,E1 -19178.377,E2 -19178.377} C_VEL
LIN {X 0,Y 241.24,Z 502.825,A -85,B 0,C 180,E1 -19180.915,E2 -19180.915} C_VEL
LIN {X 0,Y 241.751,Z 495.913,A -85,B 0,C 180,E1 -19183.448,E2 -19183.448} C_VEL
LIN {X 0,Y 242.698,Z 487.274,A -85,B 0,C 180,E1 -19185.968,E2 -19185.968} C_VEL
LIN {X 0,Y 243.996,Z 478.247,A -85,B 0,C 180,E1 -19188.098,E2 -19188.098} C_VEL
LIN {X 0,Y 244.352,Z 473.294,A -85,B 0,C 180,E1 -19189.096,E2 -19189.096} C_VEL
LIN {X 0,Y 244.363,Z 463.27,A -85,B 0,C 180,E1 -19190.849,E2 -19190.849} C_VEL
LIN {X 0,Y 244.045,Z 450.957,A -85,B 0,C 180,E1 -19192.615,E2 -19192.615} C_VEL
LIN {X 0,Y 243.578,Z 438.324,A -85,B 0,C 180,E1 -19194.05,E2 -19194.05} C_VEL
LIN {X 0,Y 242.759,Z 424.254,A -85,B 0,C 180,E1 -19195.278,E2 -19195.278} C_VEL
LIN {X 0,Y 241.912,Z 411.921,A -85,B 0,C 180,E1 -19196.136,E2 -19196.136} C_VEL
LIN {X 0,Y 243.057,Z 403.253,A -85,B 0,C 180,E1 -19200.466,E2 -19200.466} C_VEL
LIN {X 0,Y 244.7,Z 394.243,A -85,B 0,C 180,E1 -19205.058,E2 -19205.058} C_VEL
LIN {X 0,Y 245.887,Z 388.672,A -85,B 0,C 180,E1 -19207.916,E2 -19207.916} C_VEL
LIN {X 0,Y 245.974,Z 385.658,A -85,B 0,C 180,E1 -19209.516,E2 -19209.516} C_VEL
LIN {X 0,Y 244.382,Z 377.603,A -85,B 0,C 180,E1 -19214.031,E2 -19214.031} C_VEL
LIN {X 0,Y 242.942,Z 370.422,A -85,B 0,C 180,E1 -19218.29,E2 -19218.29} C_VEL
LIN {X 0,Y 242,Z 365.418,A -85,B 0,C 180,E1 -19221.409,E2 -19221.409} C_VEL
LIN {X 0,Y 241.982,Z 365.342,A -85,B 0,C 180,E1 -19224.488,E2 -19224.488} C_VEL
LIN {X 0,Y 241.971,Z 365.342,A -85,B 0,C 180,E1 -19228.479,E2 -19228.479} C_VEL
LIN {X 0,Y 242.002,Z 365.337,A -85,B 0,C 180,E1 -19232.312,E2 -19232.312} C_VEL
LIN {X 0,Y 242.035,Z 365.333,A -85,B 0,C 180,E1 -19236.014,E2 -19236.014} C_VEL
LIN {X 0,Y 242.014,Z 365.337,A -85,B 0,C 180,E1 -19239.606,E2 -19239.606} C_VEL
LIN {X 0,Y 242.111,Z 365.326,A -85,B 0,C 180,E1 -19243.316,E2 -19243.316} C_VEL
LIN {X 0,Y 242.158,Z 365.315,A -85,B 0,C 180,E1 -19248.278,E2 -19248.278} C_VEL
LIN {X 0,Y 242.382,Z 365.291,A -85,B 0,C 180,E1 -19251.664,E2 -19251.664} C_VEL
LIN {X 0,Y 242.242,Z 365.31,A -85,B 0,C 180,E1 -19255.007,E2 -19255.007} C_VEL
LIN {X 0,Y 242.628,Z 365.259,A -85,B 0,C 180,E1 -19258.34,E2 -19258.34} C_VEL
LIN {X 0,Y 242.629,Z 365.26,A -85,B 0,C 180,E1 -19261.66,E2 -19261.66} C_VEL
LIN {X 0,Y 242.416,Z 365.287,A -85,B 0,C 180,E1 -19266.803,E2 -19266.803} C_VEL
LIN {X 0,Y 242.309,Z 365.3,A -85,B 0,C 180,E1 -19270.022,E2 -19270.022} C_VEL
LIN {X 0,Y 242.158,Z 365.319,A -85,B 0,C 180,E1 -19275.141,E2 -19275.141} C_VEL
LIN {X 0,Y 242.068,Z 365.333,A -85,B 0,C 180,E1 -19278.625,E2 -19278.625} C_VEL
LIN {X 0,Y 242.008,Z 365.337,A -85,B 0,C 180,E1 -19282.18,E2 -19282.18} C_VEL
LIN {X 0,Y 242.063,Z 365.331,A -85,B 0,C 180,E1 -19285.839,E2 -19285.839} C_VEL
LIN {X 0,Y 242.026,Z 365.333,A -85,B 0,C 180,E1 -19289.581,E2 -19289.581} C_VEL
LIN {X 0,Y 241.988,Z 365.34,A -85,B 0,C 180,E1 -19293.492,E2 -19293.492} C_VEL
LIN {X 0,Y 242.008,Z 365.336,A -85,B 0,C 180,E1 -19297.579,E2 -19297.579} C_VEL
LIN {X 0,Y 241.952,Z 365.346,A -85,B 0,C 180,E1 -19301.919,E2 -19301.919} C_VEL
LIN {X 0,Y 241.932,Z 365.346,A -85,B 0,C 180,E1 -19306.572,E2 -19306.572} C_VEL
LIN {X 0,Y 241.955,Z 365.347,A -85,B 0,C 180,E1 -19310.282,E2 -19310.282} C_VEL
LIN {X 0,Y 242.036,Z 365.333,A -85,B 0,C 180,E1 -19314.498,E2 -19314.498} C_VEL
LIN {X 0,Y 241.976,Z 365.342,A -85,B 0,C 180,E1 -19318.481,E2 -19318.481} C_VEL
LIN {X 0,Y 242.012,Z 365.336,A -85,B 0,C 180,E1 -19322.314,E2 -19322.314} C_VEL
LIN {X 0,Y 242.058,Z 365.334,A -85,B 0,C 180,E1 -19326.017,E2 -19326.017} C_VEL
LIN {X 0,Y 242.039,Z 365.336,A -85,B 0,C 180,E1 -19329.609,E2 -19329.609} C_VEL
LIN {X 0,Y 242.164,Z 365.318,A -85,B 0,C 180,E1 -19333.279,E2 -19333.279} C_VEL
LIN {X 0,Y 242.188,Z 365.314,A -85,B 0,C 180,E1 -19338.28,E2 -19338.28} C_VEL
LIN {X 0,Y 242.437,Z 365.287,A -85,B 0,C 180,E1 -19341.666,E2 -19341.666} C_VEL
LIN {X 0,Y 242.264,Z 365.306,A -85,B 0,C 180,E1 -19345.007,E2 -19345.007} C_VEL
LIN {X 0,Y 242.641,Z 365.258,A -85,B 0,C 180,E1 -19348.34,E2 -19348.34} C_VEL
LIN {X 0,Y 242.639,Z 365.261,A -85,B 0,C 180,E1 -19351.66,E2 -19351.66} C_VEL
LIN {X 0,Y 242.43,Z 365.283,A -85,B 0,C 180,E1 -19356.659,E2 -19356.659} C_VEL
LIN {X 0,Y 242.314,Z 365.299,A -85,B 0,C 180,E1 -19360.021,E2 -19360.021} C_VEL
LIN {X 0,Y 242.168,Z 365.32,A -85,B 0,C 180,E1 -19365.14,E2 -19365.14} C_VEL
LIN {X 0,Y 242.074,Z 365.33,A -85,B 0,C 180,E1 -19368.624,E2 -19368.624} C_VEL
LIN {X 0,Y 242.014,Z 365.337,A -85,B 0,C 180,E1 -19372.179,E2 -19372.179} C_VEL
LIN {X 0,Y 242.067,Z 365.33,A -85,B 0,C 180,E1 -19375.837,E2 -19375.837} C_VEL
LIN {X 0,Y 242.007,Z 365.34,A -85,B 0,C 180,E1 -19379.583,E2 -19379.583} C_VEL
LIN {X 0,Y 241.99,Z 365.342,A -85,B 0,C 180,E1 -19383.49,E2 -19383.49} C_VEL
LIN {X 0,Y 242.076,Z 365.478,A -85,B 0,C 180,E1 -19387.565,E2 -19387.565} C_VEL
LIN {X 0,Y 242.349,Z 366.641,A -85,B 0,C 180,E1 -19387.883,E2 -19387.883} C_VEL
LIN {X 0,Y 246.101,Z 379.36,A -85,B 0,C 180,E1 -19389.552,E2 -19389.552} C_VEL
LIN {X 0,Y 249.008,Z 390.392,A -85,B 0,C 180,E1 -19391.278,E2 -19391.278} C_VEL
LIN {X 0,Y 249.278,Z 392.731,A -85,B 0,C 180,E1 -19391.658,E2 -19391.658} C_VEL
LIN {X 0,Y 247.944,Z 403.38,A -85,B 0,C 180,E1 -19393.445,E2 -19393.445} C_VEL
LIN {X 0,Y 246.615,Z 413.034,A -85,B 0,C 180,E1 -19395.433,E2 -19395.433} C_VEL
LIN {X 0,Y 245.436,Z 421.347,A -85,B 0,C 180,E1 -19397.509,E2 -19397.509} C_VEL
LIN {X 0,Y 244.484,Z 428.611,A -85,B 0,C 180,E1 -19399.7,E2 -19399.7} C_VEL
LIN {X 0,Y 243.641,Z 434.598,A -85,B 0,C 180,E1 -19401.876,E2 -19401.876} C_VEL
LIN {X 0,Y 242.986,Z 440.757,A -85,B 0,C 180,E1 -19404.657,E2 -19404.657} C_VEL
LIN {X 0,Y 242.59,Z 445.063,A -85,B 0,C 180,E1 -19407.154,E2 -19407.154} C_VEL
LIN {X 0,Y 242.441,Z 449.148,A -85,B 0,C 180,E1 -19410.416,E2 -19410.416} C_VEL
LIN {X 0,Y 242.575,Z 450.83,A -85,B 0,C 180,E1 -19412.383,E2 -19412.383} C_VEL
LIN {X 0,Y 242.91,Z 451.921,A -85,B 0,C 180,E1 -19414.279,E2 -19414.279} C_VEL
LIN {X 0,Y 243.766,Z 452.614,A -85,B 0,C 180,E1 -19417.304,E2 -19417.304} C_VEL
LIN {X 0,Y 244.848,Z 452.164,A -85,B 0,C 180,E1 -19419.852,E2 -19419.852} C_VEL
LIN {X 0,Y 245.791,Z 451.243,A -85,B 0,C 180,E1 -19421.668,E2 -19421.668} C_VEL
LIN {X 0,Y 247.742,Z 448.639,A -85,B 0,C 180,E1 -19424.687,E2 -19424.687} C_VEL
LIN {X 0,Y 249.625,Z 445.59,A -85,B 0,C 180,E1 -19426.983,E2 -19426.983} C_VEL
LIN {X 0,Y 252.199,Z 440.968,A -85,B 0,C 180,E1 -19429.564,E2 -19429.564} C_VEL
LIN {X 0,Y 255.303,Z 434.402,A -85,B 0,C 180,E1 -19432.302,E2 -19432.302} C_VEL
LIN {X 0,Y 258.264,Z 427.465,A -85,B 0,C 180,E1 -19434.535,E2 -19434.535} C_VEL
LIN {X 0,Y 261.173,Z 419.783,A -85,B 0,C 180,E1 -19436.52,E2 -19436.52} C_VEL
LIN {X 0,Y 263.128,Z 414.085,A -85,B 0,C 180,E1 -19437.753,E2 -19437.753} C_VEL
LIN {X 0,Y 263.377,Z 412.588,A -85,B 0,C 180,E1 -19438.113,E2 -19438.113} C_VEL
LIN {X 0,Y 262.218,Z 406.318,A -85,B 0,C 180,E1 -19440,E2 -19440} C_VEL
LIN {X 0,Y 260.081,Z 397.297,A -85,B 0,C 180,E1 -19442.602,E2 -19442.602} C_VEL
LIN {X 0,Y 257.361,Z 390.59,A -85,B 0,C 180,E1 -19444.699,E2 -19444.699} C_VEL
LIN {X 0,Y 252.481,Z 381.068,A -85,B 0,C 180,E1 -19448,E2 -19448} C_VEL
LIN {X 0,Y 249.649,Z 376.245,A -85,B 0,C 180,E1 -19449.843,E2 -19449.843} C_VEL
LIN {X 0,Y 246.751,Z 372.577,A -85,B 0,C 180,E1 -19451.605,E2 -19451.605} C_VEL
LIN {X 0,Y 245.86,Z 370.74,A -85,B 0,C 180,E1 -19452.276,E2 -19452.276} C_VEL
LIN {X 0,Y 243.301,Z 368.462,A -85,B 0,C 180,E1 -19453.84,E2 -19453.84} C_VEL
LIN {X 0,Y 242.594,Z 367.118,A -85,B 0,C 180,E1 -19454.47,E2 -19454.47} C_VEL
LIN {X 0,Y 242.437,Z 366.713,A -85,B 0,C 180,E1 -19455.124,E2 -19455.124} C_VEL
LIN {X 0,Y 242.501,Z 367.455,A -85,B 0,C 180,E1 -19458.59,E2 -19458.59} C_VEL
LIN {X 0,Y 242.741,Z 368.614,A -85,B 0,C 180,E1 -19462.11,E2 -19462.11} C_VEL
LIN {X 0,Y 243.277,Z 370.586,A -85,B 0,C 180,E1 -19466.423,E2 -19466.423} C_VEL
LIN {X 0,Y 243.723,Z 372.866,A -85,B 0,C 180,E1 -19470.111,E2 -19470.111} C_VEL
LIN {X 0,Y 244.235,Z 375.384,A -85,B 0,C 180,E1 -19473.439,E2 -19473.439} C_VEL
LIN {X 0,Y 244.906,Z 378.612,A -85,B 0,C 180,E1 -19477.059,E2 -19477.059} C_VEL
LIN {X 0,Y 245.836,Z 382.848,A -85,B 0,C 180,E1 -19481.112,E2 -19481.112} C_VEL
LIN {X 0,Y 246.133,Z 384.42,A -85,B 0,C 180,E1 -19482.456,E2 -19482.456} C_VEL
LIN {X 0,Y 245.617,Z 385.721,A -85,B 0,C 180,E1 -19483.349,E2 -19483.349} C_VEL
LIN {X 0,Y 243.01,Z 388.302,A -85,B 0,C 180,E1 -19484.725,E2 -19484.725} C_VEL
LIN {X 0,Y 240.842,Z 391.344,A -85,B 0,C 180,E1 -19486.046,E2 -19486.046} C_VEL
LIN {X 0,Y 240.956,Z 393.521,A -85,B 0,C 180,E1 -19486.821,E2 -19486.821} C_VEL
LIN {X 0,Y 243.682,Z 398.732,A -85,B 0,C 180,E1 -19488.579,E2 -19488.579} C_VEL
LIN {X 0,Y 244.343,Z 400.34,A -85,B 0,C 180,E1 -19489.024,E2 -19489.024} C_VEL
LIN {X 0,Y 245.863,Z 405.958,A -85,B 0,C 180,E1 -19490.267,E2 -19490.267} C_VEL
LIN {X 0,Y 247.62,Z 414.822,A -85,B 0,C 180,E1 -19492.003,E2 -19492.003} C_VEL
LIN {X 0,Y 249.401,Z 428.757,A -85,B 0,C 180,E1 -19494.562,E2 -19494.562} C_VEL
LIN {X 0,Y 249.956,Z 441.111,A -85,B 0,C 180,E1 -19496.772,E2 -19496.772} C_VEL
LIN {X 0,Y 249.286,Z 454.372,A -85,B 0,C 180,E1 -19499.206,E2 -19499.206} C_VEL
LIN {X 0,Y 247.933,Z 464.395,A -85,B 0,C 180,E1 -19501.192,E2 -19501.192} C_VEL
LIN {X 0,Y 245.326,Z 475.581,A -85,B 0,C 180,E1 -19503.639,E2 -19503.639} C_VEL
LIN {X 0,Y 242.616,Z 484.907,A -85,B 0,C 180,E1 -19506.075,E2 -19506.075} C_VEL
LIN {X 0,Y 239.774,Z 492.702,A -85,B 0,C 180,E1 -19508.508,E2 -19508.508} C_VEL
LIN {X 0,Y 237.002,Z 500.265,A -85,B 0,C 180,E1 -19511.435,E2 -19511.435} C_VEL
LIN {X 0,Y 235.143,Z 506.183,A -85,B 0,C 180,E1 -19514.396,E2 -19514.396} C_VEL
LIN {X 0,Y 233.846,Z 511.332,A -85,B 0,C 180,E1 -19517.856,E2 -19517.856} C_VEL
LIN {X 0,Y 233.593,Z 513.326,A -85,B 0,C 180,E1 -19519.6,E2 -19519.6} C_VEL
LIN {X 0,Y 233.798,Z 516.09,A -85,B 0,C 180,E1 -19523.094,E2 -19523.094} C_VEL
LIN {X 0,Y 234.096,Z 516.884,A -85,B 0,C 180,E1 -19524.833,E2 -19524.833} C_VEL
LIN {X 0,Y 234.99,Z 517.289,A -85,B 0,C 180,E1 -19528.286,E2 -19528.286} C_VEL
LIN {X 0,Y 235.466,Z 516.827,A -85,B 0,C 180,E1 -19530,E2 -19530} C_VEL
LIN {X 0,Y 235.108,Z 515.778,A -85,B 0,C 180,E1 -19531.713,E2 -19531.713} C_VEL
LIN {X 0,Y 234.778,Z 514.284,A -85,B 0,C 180,E1 -19533.432,E2 -19533.432} C_VEL
LIN {X 0,Y 234.492,Z 511.123,A -85,B 0,C 180,E1 -19536.021,E2 -19536.021} C_VEL
LIN {X 0,Y 234.134,Z 506.741,A -85,B 0,C 180,E1 -19538.632,E2 -19538.632} C_VEL
LIN {X 0,Y 234.317,Z 500.006,A -85,B 0,C 180,E1 -19541.68,E2 -19541.68} C_VEL
LIN {X 0,Y 234.931,Z 492.663,A -85,B 0,C 180,E1 -19544.288,E2 -19544.288} C_VEL
LIN {X 0,Y 235.86,Z 485.193,A -85,B 0,C 180,E1 -19546.443,E2 -19546.443} C_VEL
LIN {X 0,Y 237.262,Z 475.412,A -85,B 0,C 180,E1 -19548.729,E2 -19548.729} C_VEL
LIN {X 0,Y 237.328,Z 464.455,A -85,B 0,C 180,E1 -19550.815,E2 -19550.815} C_VEL
LIN {X 0,Y 237.041,Z 452.415,A -85,B 0,C 180,E1 -19552.67,E2 -19552.67} C_VEL
LIN {X 0,Y 236.681,Z 440.337,A -85,B 0,C 180,E1 -19554.162,E2 -19554.162} C_VEL
LIN {X 0,Y 235.965,Z 427.249,A -85,B 0,C 180,E1 -19555.436,E2 -19555.436} C_VEL
LIN {X 0,Y 234.919,Z 411.111,A -85,B 0,C 180,E1 -19556.619,E2 -19556.619} C_VEL
LIN {X 0,Y 235.67,Z 405.617,A -85,B 0,C 180,E1 -19559.375,E2 -19559.375} C_VEL
LIN {X 0,Y 237.29,Z 396.361,A -85,B 0,C 180,E1 -19564.244,E2 -19564.244} C_VEL
LIN {X 0,Y 238.875,Z 389.002,A -85,B 0,C 180,E1 -19568.158,E2 -19568.158} C_VEL
LIN {X 0,Y 239.024,Z 387.345,A -85,B 0,C 180,E1 -19569.059,E2 -19569.059} C_VEL
LIN {X 0,Y 237.793,Z 380.735,A -85,B 0,C 180,E1 -19572.824,E2 -19572.824} C_VEL
LIN {X 0,Y 236.176,Z 372.819,A -85,B 0,C 180,E1 -19577.58,E2 -19577.58} C_VEL
LIN {X 0,Y 234.985,Z 366.283,A -85,B 0,C 180,E1 -19581.777,E2 -19581.777} C_VEL
LIN {X 0,Y 234.939,Z 366.22,A -85,B 0,C 180,E1 -19586.885,E2 -19586.885} C_VEL
LIN {X 0,Y 234.947,Z 366.219,A -85,B 0,C 180,E1 -19591.405,E2 -19591.405} C_VEL
LIN {X 0,Y 234.973,Z 366.216,A -85,B 0,C 180,E1 -19595.245,E2 -19595.245} C_VEL
LIN {X 0,Y 234.984,Z 366.213,A -85,B 0,C 180,E1 -19598.967,E2 -19598.967} C_VEL
LIN {X 0,Y 235.051,Z 366.207,A -85,B 0,C 180,E1 -19603.092,E2 -19603.092} C_VEL
LIN {X 0,Y 235.091,Z 366.195,A -85,B 0,C 180,E1 -19607.921,E2 -19607.921} C_VEL
LIN {X 0,Y 235.311,Z 366.173,A -85,B 0,C 180,E1 -19611.412,E2 -19611.412} C_VEL
LIN {X 0,Y 235.357,Z 366.168,A -85,B 0,C 180,E1 -19613.14,E2 -19613.14} C_VEL
LIN {X 0,Y 235.588,Z 366.136,A -85,B 0,C 180,E1 -19618.29,E2 -19618.29} C_VEL
LIN {X 0,Y 235.588,Z 366.137,A -85,B 0,C 180,E1 -19621.709,E2 -19621.709} C_VEL
LIN {X 0,Y 235.396,Z 366.164,A -85,B 0,C 180,E1 -19626.859,E2 -19626.859} C_VEL
LIN {X 0,Y 235.233,Z 366.183,A -85,B 0,C 180,E1 -19630.327,E2 -19630.327} C_VEL
LIN {X 0,Y 235.107,Z 366.196,A -85,B 0,C 180,E1 -19635.607,E2 -19635.607} C_VEL
LIN {X 0,Y 235.004,Z 366.21,A -85,B 0,C 180,E1 -19639.206,E2 -19639.206} C_VEL
LIN {X 0,Y 234.956,Z 366.216,A -85,B 0,C 180,E1 -19642.883,E2 -19642.883} C_VEL
LIN {X 0,Y 234.966,Z 366.217,A -85,B 0,C 180,E1 -19646.658,E2 -19646.658} C_VEL
LIN {X 0,Y 234.928,Z 366.221,A -85,B 0,C 180,E1 -19650.568,E2 -19650.568} C_VEL
LIN {X 0,Y 234.957,Z 366.217,A -85,B 0,C 180,E1 -19654.634,E2 -19654.634} C_VEL
LIN {X 0,Y 234.964,Z 366.213,A -85,B 0,C 180,E1 -19658.953,E2 -19658.953} C_VEL
LIN {X 0,Y 234.917,Z 366.221,A -85,B 0,C 180,E1 -19663.479,E2 -19663.479} C_VEL
LIN {X 0,Y 234.886,Z 366.224,A -85,B 0,C 180,E1 -19666.515,E2 -19666.515} C_VEL
LIN {X 0,Y 234.918,Z 366.22,A -85,B 0,C 180,E1 -19671.08,E2 -19671.08} C_VEL
LIN {X 0,Y 234.959,Z 366.213,A -85,B 0,C 180,E1 -19675.368,E2 -19675.368} C_VEL
LIN {X 0,Y 234.97,Z 366.216,A -85,B 0,C 180,E1 -19680.158,E2 -19680.158} C_VEL
LIN {X 0,Y 234.995,Z 366.211,A -85,B 0,C 180,E1 -19683.794,E2 -19683.794} C_VEL
LIN {X 0,Y 235.012,Z 366.208,A -85,B 0,C 180,E1 -19688.971,E2 -19688.971} C_VEL
LIN {X 0,Y 235.098,Z 366.197,A -85,B 0,C 180,E1 -19693.06,E2 -19693.06} C_VEL
LIN {X 0,Y 235.148,Z 366.192,A -85,B 0,C 180,E1 -19697.924,E2 -19697.924} C_VEL
LIN {X 0,Y 235.392,Z 366.162,A -85,B 0,C 180,E1 -19701.415,E2 -19701.415} C_VEL
LIN {X 0,Y 235.408,Z 366.161,A -85,B 0,C 180,E1 -19703.142,E2 -19703.142} C_VEL
LIN {X 0,Y 235.601,Z 366.135,A -85,B 0,C 180,E1 -19708.291,E2 -19708.291} C_VEL
LIN {X 0,Y 235.599,Z 366.137,A -85,B 0,C 180,E1 -19711.709,E2 -19711.709} C_VEL
LIN {X 0,Y 235.4,Z 366.159,A -85,B 0,C 180,E1 -19716.859,E2 -19716.859} C_VEL
LIN {X 0,Y 235.239,Z 366.18,A -85,B 0,C 180,E1 -19720.326,E2 -19720.326} C_VEL
LIN {X 0,Y 235.115,Z 366.198,A -85,B 0,C 180,E1 -19725.606,E2 -19725.606} C_VEL
LIN {X 0,Y 235.01,Z 366.213,A -85,B 0,C 180,E1 -19729.205,E2 -19729.205} C_VEL
LIN {X 0,Y 234.962,Z 366.218,A -85,B 0,C 180,E1 -19732.882,E2 -19732.882} C_VEL
LIN {X 0,Y 234.968,Z 366.215,A -85,B 0,C 180,E1 -19736.657,E2 -19736.657} C_VEL
LIN {X 0,Y 234.922,Z 366.222,A -85,B 0,C 180,E1 -19740.568,E2 -19740.568} C_VEL
LIN {X 0,Y 234.96,Z 366.219,A -85,B 0,C 180,E1 -19744.632,E2 -19744.632} C_VEL
LIN {X 0,Y 235.039,Z 366.395,A -85,B 0,C 180,E1 -19747.13,E2 -19747.13} C_VEL
LIN {X 0,Y 235.386,Z 367.765,A -85,B 0,C 180,E1 -19747.469,E2 -19747.469} C_VEL
LIN {X 0,Y 239.139,Z 380.602,A -85,B 0,C 180,E1 -19749.213,E2 -19749.213} C_VEL
LIN {X 0,Y 242.175,Z 392.198,A -85,B 0,C 180,E1 -19751.096,E2 -19751.096} C_VEL
LIN {X 0,Y 242.364,Z 393.593,A -85,B 0,C 180,E1 -19751.33,E2 -19751.33} C_VEL
LIN {X 0,Y 240.971,Z 404.346,A -85,B 0,C 180,E1 -19753.186,E2 -19753.186} C_VEL
LIN {X 0,Y 239.44,Z 415.2,A -85,B 0,C 180,E1 -19755.511,E2 -19755.511} C_VEL
LIN {X 0,Y 238.129,Z 424.246,A -85,B 0,C 180,E1 -19757.917,E2 -19757.917} C_VEL
LIN {X 0,Y 237.084,Z 431.865,A -85,B 0,C 180,E1 -19760.418,E2 -19760.418} C_VEL
LIN {X 0,Y 236.264,Z 438.163,A -85,B 0,C 180,E1 -19762.961,E2 -19762.961} C_VEL
LIN {X 0,Y 235.713,Z 443.199,A -85,B 0,C 180,E1 -19765.493,E2 -19765.493} C_VEL
LIN {X 0,Y 235.434,Z 447.795,A -85,B 0,C 180,E1 -19768.507,E2 -19768.507} C_VEL
LIN {X 0,Y 235.458,Z 450.96,A -85,B 0,C 180,E1 -19771.473,E2 -19771.473} C_VEL
LIN {X 0,Y 235.687,Z 452.414,A -85,B 0,C 180,E1 -19773.451,E2 -19773.451} C_VEL
LIN {X 0,Y 236.135,Z 453.297,A -85,B 0,C 180,E1 -19775.375,E2 -19775.375} C_VEL
LIN {X 0,Y 236.729,Z 453.691,A -85,B 0,C 180,E1 -19777.298,E2 -19777.298} C_VEL
LIN {X 0,Y 237.523,Z 453.605,A -85,B 0,C 180,E1 -19779.203,E2 -19779.203} C_VEL
LIN {X 0,Y 238.43,Z 453.003,A -85,B 0,C 180,E1 -19781.081,E2 -19781.081} C_VEL
LIN {X 0,Y 239.548,Z 451.953,A -85,B 0,C 180,E1 -19782.939,E2 -19782.939} C_VEL
LIN {X 0,Y 241.493,Z 449.462,A -85,B 0,C 180,E1 -19785.678,E2 -19785.678} C_VEL
LIN {X 0,Y 243.929,Z 445.726,A -85,B 0,C 180,E1 -19788.399,E2 -19788.399} C_VEL
LIN {X 0,Y 246.731,Z 440.838,A -85,B 0,C 180,E1 -19790.987,E2 -19790.987} C_VEL
LIN {X 0,Y 249.824,Z 434.568,A -85,B 0,C 180,E1 -19793.539,E2 -19793.539} C_VEL
LIN {X 0,Y 253.138,Z 427.176,A -85,B 0,C 180,E1 -19795.879,E2 -19795.879} C_VEL
LIN {X 0,Y 256.577,Z 418.505,A -85,B 0,C 180,E1 -19798.038,E2 -19798.038} C_VEL
LIN {X 0,Y 257.464,Z 415.289,A -85,B 0,C 180,E1 -19798.793,E2 -19798.793} C_VEL
LIN {X 0,Y 255.751,Z 405.279,A -85,B 0,C 180,E1 -19801.97,E2 -19801.97} C_VEL
LIN {X 0,Y 254.202,Z 399.348,A -85,B 0,C 180,E1 -19803.825,E2 -19803.825} C_VEL
LIN {X 0,Y 251.67,Z 393.242,A -85,B 0,C 180,E1 -19805.985,E2 -19805.985} C_VEL
LIN {X 0,Y 247.468,Z 384.775,A -85,B 0,C 180,E1 -19809.216,E2 -19809.216} C_VEL
LIN {X 0,Y 245.932,Z 381.956,A -85,B 0,C 180,E1 -19810.362,E2 -19810.362} C_VEL
LIN {X 0,Y 243.394,Z 378.305,A -85,B 0,C 180,E1 -19812.19,E2 -19812.19} C_VEL
LIN {X 0,Y 242.879,Z 377.078,A -85,B 0,C 180,E1 -19812.652,E2 -19812.652} C_VEL
LIN {X 0,Y 240.456,Z 374.587,A -85,B 0,C 180,E1 -19814.353,E2 -19814.353} C_VEL
LIN {X 0,Y 239.615,Z 373.214,A -85,B 0,C 180,E1 -19815.081,E2 -19815.081} C_VEL
LIN {X 0,Y 237.099,Z 371.649,A -85,B 0,C 180,E1 -19816.933,E2 -19816.933} C_VEL
LIN {X 0,Y 235.946,Z 370.066,A -85,B 0,C 180,E1 -19818.227,E2 -19818.227} C_VEL
LIN {X 0,Y 235.825,Z 369.961,A -85,B 0,C 180,E1 -19819.137,E2 -19819.137} C_VEL
LIN {X 0,Y 236.067,Z 371.224,A -85,B 0,C 180,E1 -19822.77,E2 -19822.77} C_VEL
LIN {X 0,Y 236.645,Z 373.245,A -85,B 0,C 180,E1 -19827.009,E2 -19827.009} C_VEL
LIN {X 0,Y 237.087,Z 375.617,A -85,B 0,C 180,E1 -19830.725,E2 -19830.725} C_VEL
LIN {X 0,Y 237.612,Z 378.26,A -85,B 0,C 180,E1 -19834.193,E2 -19834.193} C_VEL
LIN {X 0,Y 238.407,Z 381.953,A -85,B 0,C 180,E1 -19838.248,E2 -19838.248} C_VEL
LIN {X 0,Y 239.353,Z 386.494,A -85,B 0,C 180,E1 -19842.481,E2 -19842.481} C_VEL
LIN {X 0,Y 240.225,Z 391.071,A -85,B 0,C 180,E1 -19846.009,E2 -19846.009} C_VEL
LIN {X 0,Y 240.773,Z 393.025,A -85,B 0,C 180,E1 -19846.677,E2 -19846.677} C_VEL
LIN {X 0,Y 240.956,Z 393.521,A -85,B 0,C 180,E1 -19846.821,E2 -19846.821} C_VEL
LIN {X 0,Y 242.123,Z 397.521,A -85,B 0,C 180,E1 -19847.816,E2 -19847.816} C_VEL
LIN {X 0,Y 242.708,Z 402.288,A -85,B 0,C 180,E1 -19848.648,E2 -19848.648} C_VEL
LIN {X 0,Y 242.784,Z 416.029,A -85,B 0,C 180,E1 -19850.664,E2 -19850.664} C_VEL
LIN {X 0,Y 242.991,Z 419.215,A -85,B 0,C 180,E1 -19851.252,E2 -19851.252} C_VEL
LIN {X 0,Y 244.115,Z 431.812,A -85,B 0,C 180,E1 -19853.718,E2 -19853.718} C_VEL
LIN {X 0,Y 244.235,Z 443.822,A -85,B 0,C 180,E1 -19856.025,E2 -19856.025} C_VEL
LIN {X 0,Y 243.311,Z 455.563,A -85,B 0,C 180,E1 -19858.341,E2 -19858.341} C_VEL
LIN {X 0,Y 241.493,Z 466.549,A -85,B 0,C 180,E1 -19860.666,E2 -19860.666} C_VEL
LIN {X 0,Y 238.488,Z 477.59,A -85,B 0,C 180,E1 -19863.295,E2 -19863.295} C_VEL
LIN {X 0,Y 235.159,Z 487.67,A -85,B 0,C 180,E1 -19866.206,E2 -19866.206} C_VEL
LIN {X 0,Y 231.813,Z 495.892,A -85,B 0,C 180,E1 -19869.132,E2 -19869.132} C_VEL
LIN {X 0,Y 229.229,Z 502.465,A -85,B 0,C 180,E1 -19872.146,E2 -19872.146} C_VEL
LIN {X 0,Y 227.446,Z 508.305,A -85,B 0,C 180,E1 -19875.689,E2 -19875.689} C_VEL
LIN {X 0,Y 226.843,Z 510.609,A -85,B 0,C 180,E1 -19877.475,E2 -19877.475} C_VEL
LIN {X 0,Y 226.479,Z 513.978,A -85,B 0,C 180,E1 -19881.074,E2 -19881.074} C_VEL
LIN {X 0,Y 227.029,Z 515.86,A -85,B 0,C 180,E1 -19884.671,E2 -19884.671} C_VEL
LIN {X 0,Y 227.368,Z 516.185,A -85,B 0,C 180,E1 -19886.456,E2 -19886.456} C_VEL
LIN {X 0,Y 227.942,Z 516.098,A -85,B 0,C 180,E1 -19888.233,E2 -19888.233} C_VEL
LIN {X 0,Y 228.46,Z 515.585,A -85,B 0,C 180,E1 -19890,E2 -19890} C_VEL
LIN {X 0,Y 228.076,Z 514.483,A -85,B 0,C 180,E1 -19891.766,E2 -19891.766} C_VEL
LIN {X 0,Y 227.656,Z 511.939,A -85,B 0,C 180,E1 -19894.426,E2 -19894.426} C_VEL
LIN {X 0,Y 227.279,Z 508.253,A -85,B 0,C 180,E1 -19897.105,E2 -19897.105} C_VEL
LIN {X 0,Y 227.086,Z 503.343,A -85,B 0,C 180,E1 -19899.8,E2 -19899.8} C_VEL
LIN {X 0,Y 227.412,Z 497.102,A -85,B 0,C 180,E1 -19902.493,E2 -19902.493} C_VEL
LIN {X 0,Y 228.152,Z 489.259,A -85,B 0,C 180,E1 -19905.179,E2 -19905.179} C_VEL
LIN {X 0,Y 229.235,Z 481.307,A -85,B 0,C 180,E1 -19907.392,E2 -19907.392} C_VEL
LIN {X 0,Y 230.158,Z 475.32,A -85,B 0,C 180,E1 -19908.808,E2 -19908.808} C_VEL
LIN {X 0,Y 230.23,Z 464.208,A -85,B 0,C 180,E1 -19911.019,E2 -19911.019} C_VEL
LIN {X 0,Y 229.989,Z 452.428,A -85,B 0,C 180,E1 -19912.93,E2 -19912.93} C_VEL
